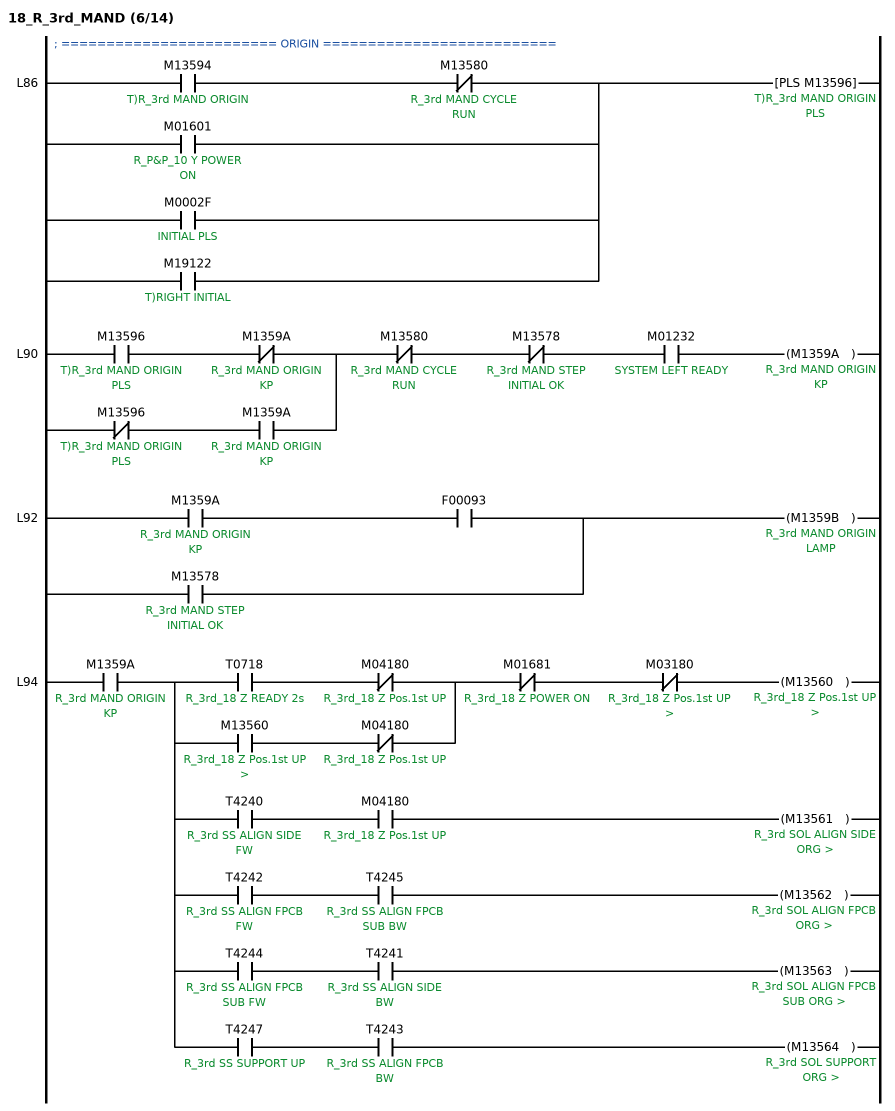
[picture p168: 18_R_3rd_MAND rungs L86-L94]
// ======================== ORIGIN ==========================
; L86
LOAD      M13594	// T)R_3rd MAND ORIGIN
AND NOT   M13580	// R_3rd MAND CYCLE RUN
OR        M01601	// R_P&P_10 Y POWER ON
OR        M0002F	// INITIAL PLS
OR        M19122	// T)RIGHT INITIAL
OUTP      M13596	// T)R_3rd MAND ORIGIN PLS
; L90
LOAD      M13596	// T)R_3rd MAND ORIGIN PLS
AND NOT   M1359A	// R_3rd MAND ORIGIN KP
LOAD NOT  M13596	// T)R_3rd MAND ORIGIN PLS
AND       M1359A	// R_3rd MAND ORIGIN KP
OR LOAD
AND NOT   M13580	// R_3rd MAND CYCLE RUN
AND NOT   M13578	// R_3rd MAND STEP INITIAL OK
AND       M01232	// SYSTEM LEFT READY
OUT       M1359A	// R_3rd MAND ORIGIN KP
; L92
LOAD      M1359A	// R_3rd MAND ORIGIN KP
AND       F00093
OR        M13578	// R_3rd MAND STEP INITIAL OK
OUT       M1359B	// R_3rd MAND ORIGIN LAMP
; L94
LOAD      M1359A	// R_3rd MAND ORIGIN KP
MPUSH
LOAD      T0718	// R_3rd_18 Z READY 2s
AND NOT   M04180	// R_3rd_18 Z Pos.1st UP
LOAD      M13560	// R_3rd_18 Z Pos.1st UP >
AND NOT   M04180	// R_3rd_18 Z Pos.1st UP
OR LOAD
AND LOAD
AND NOT   M01681	// R_3rd_18 Z POWER ON
AND NOT   M03180	// R_3rd_18 Z Pos.1st UP >
OUT       M13560	// R_3rd_18 Z Pos.1st UP >
MLOAD
AND       T4240	// R_3rd SS ALIGN SIDE FW
AND       M04180	// R_3rd_18 Z Pos.1st UP
OUT       M13561	// R_3rd SOL ALIGN SIDE ORG >
MLOAD
AND       T4242	// R_3rd SS ALIGN FPCB FW
AND       T4245	// R_3rd SS ALIGN FPCB SUB BW
OUT       M13562	// R_3rd SOL ALIGN FPCB ORG >
MLOAD
AND       T4244	// R_3rd SS ALIGN FPCB SUB FW
AND       T4241	// R_3rd SS ALIGN SIDE BW
OUT       M13563	// R_3rd SOL ALIGN FPCB SUB ORG >
MPOP
AND       T4247	// R_3rd SS SUPPORT UP
AND       T4243	// R_3rd SS ALIGN FPCB BW
OUT       M13564	// R_3rd SOL SUPPORT ORG >

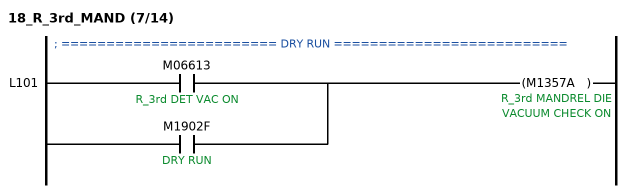
// ======================== DRY RUN ==========================
; L101
LOAD      M06613	// R_3rd DET VAC ON
OR        M1902F	// DRY RUN
OUT       M1357A	// R_3rd MANDREL DIE VACUUM CHECK ON

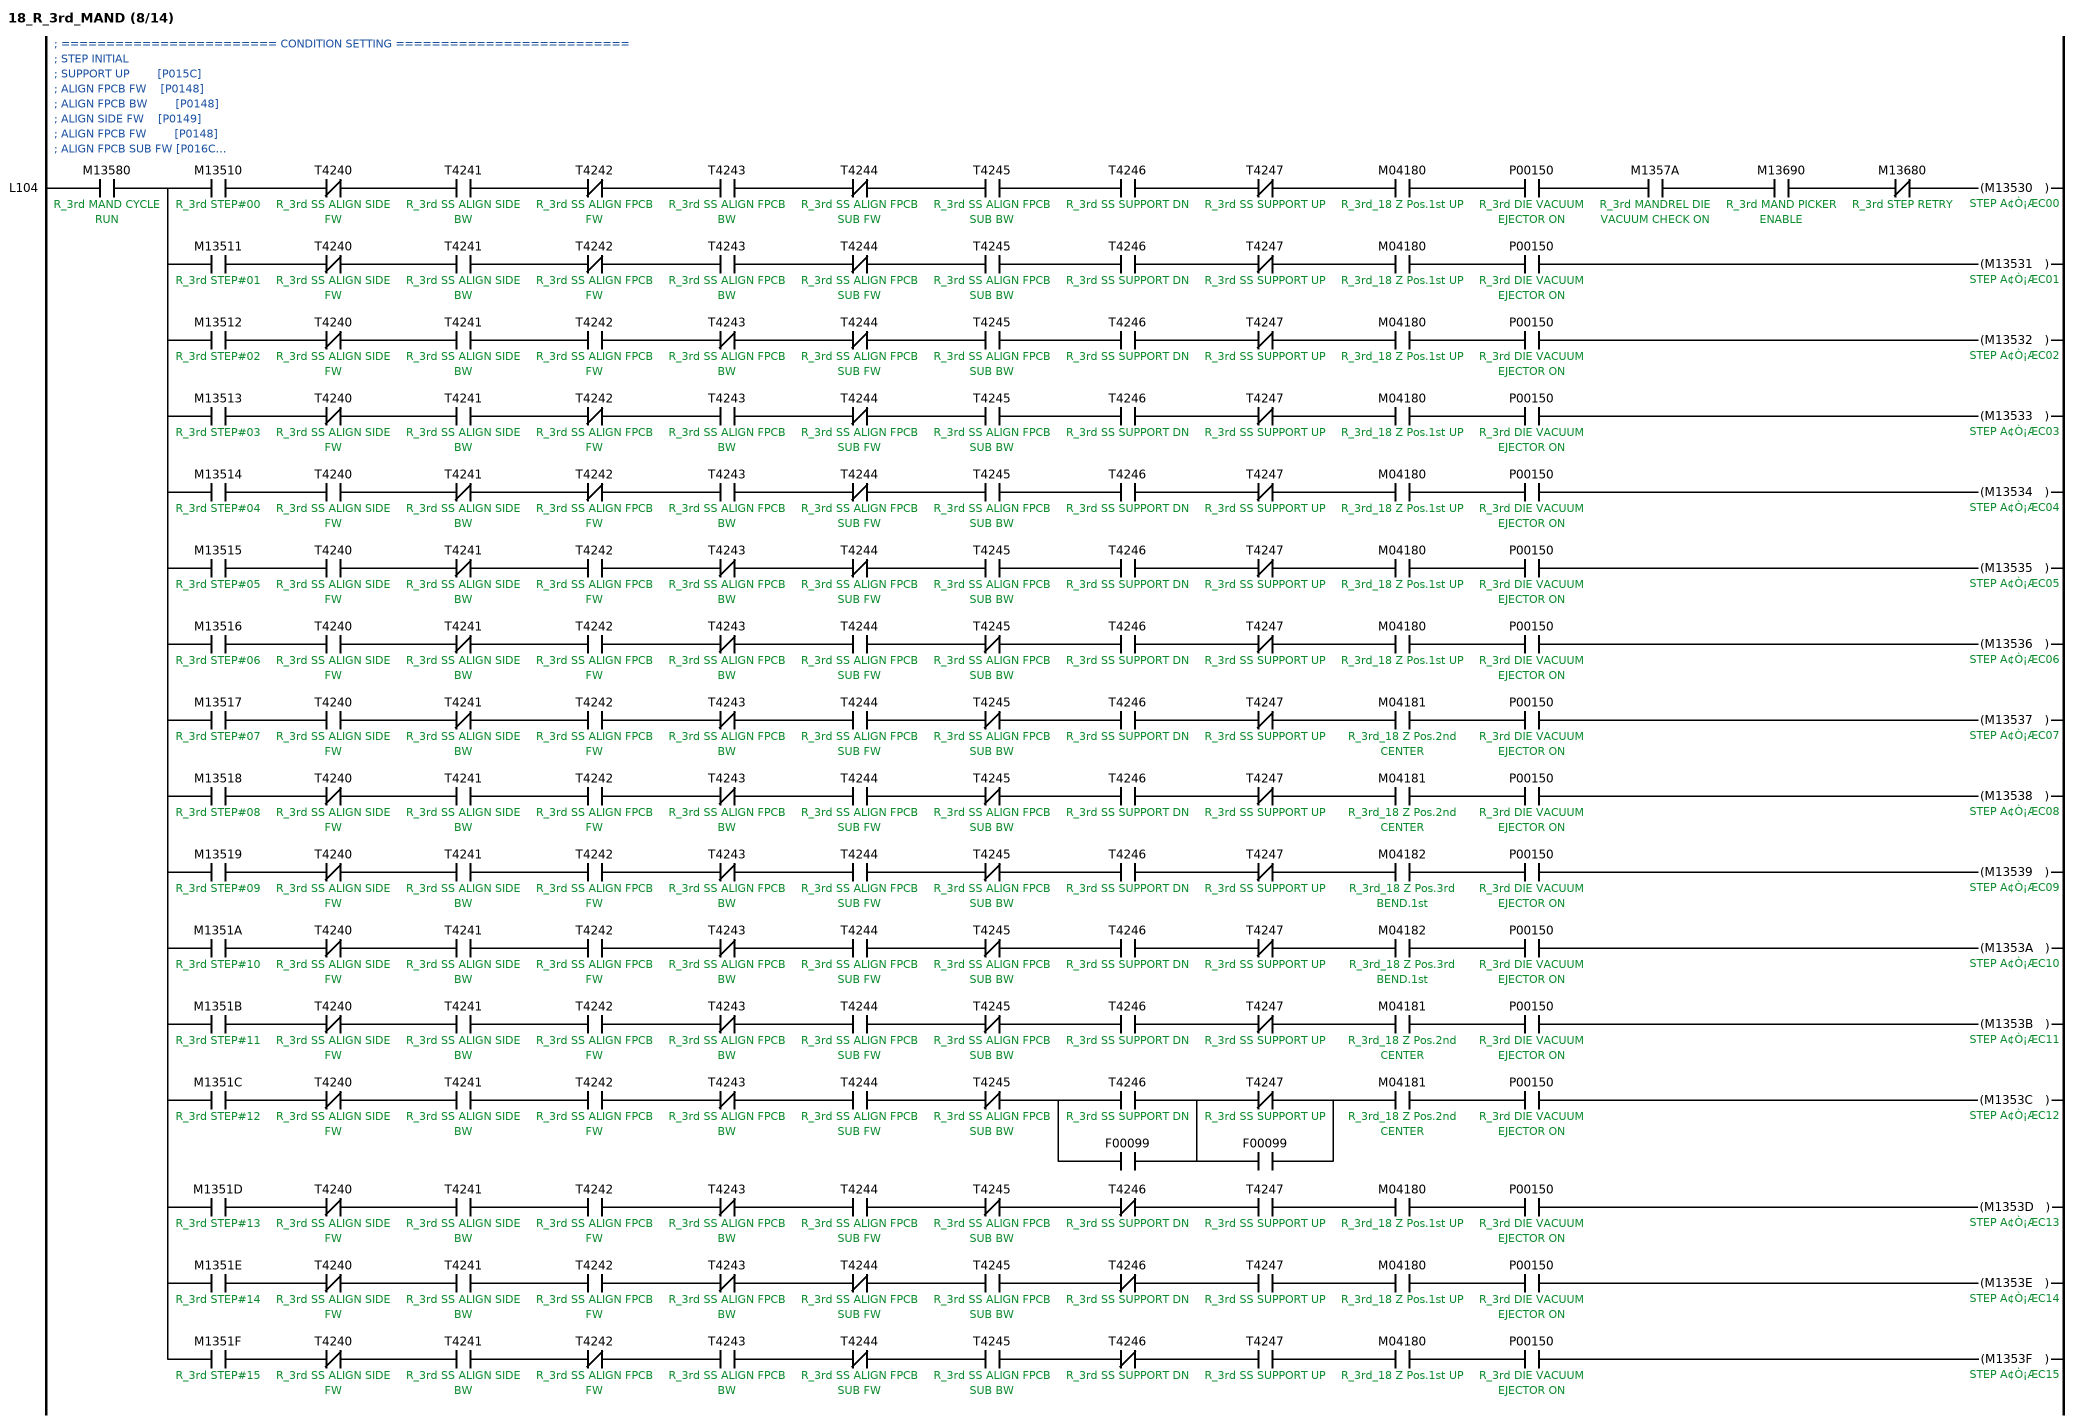
// ======================== CONDITION SETTING ==========================
; L104
LOAD      M13580	// R_3rd MAND CYCLE RUN
MPUSH
AND       M13510	// R_3rd STEP#00
AND NOT   T4240	// R_3rd SS ALIGN SIDE FW
AND       T4241	// R_3rd SS ALIGN SIDE BW
AND NOT   T4242	// R_3rd SS ALIGN FPCB FW
AND       T4243	// R_3rd SS ALIGN FPCB BW
AND NOT   T4244	// R_3rd SS ALIGN FPCB SUB FW
AND       T4245	// R_3rd SS ALIGN FPCB SUB BW
AND       T4246	// R_3rd SS SUPPORT DN
AND NOT   T4247	// R_3rd SS SUPPORT UP
AND       M04180	// R_3rd_18 Z Pos.1st UP
AND       P00150	// R_3rd DIE VACUUM EJECTOR ON
AND       M1357A	// R_3rd MANDREL DIE VACUUM CHECK ON
AND       M13690	// R_3rd MAND PICKER ENABLE
AND NOT   M13680	// R_3rd STEP RETRY
OUT       M13530	// STEP A¢Ò¡ÆC00
MLOAD
AND       M13511	// R_3rd STEP#01
AND NOT   T4240	// R_3rd SS ALIGN SIDE FW
AND       T4241	// R_3rd SS ALIGN SIDE BW
AND NOT   T4242	// R_3rd SS ALIGN FPCB FW
AND       T4243	// R_3rd SS ALIGN FPCB BW
AND NOT   T4244	// R_3rd SS ALIGN FPCB SUB FW
AND       T4245	// R_3rd SS ALIGN FPCB SUB BW
AND       T4246	// R_3rd SS SUPPORT DN
AND NOT   T4247	// R_3rd SS SUPPORT UP
AND       M04180	// R_3rd_18 Z Pos.1st UP
AND       P00150	// R_3rd DIE VACUUM EJECTOR ON
OUT       M13531	// STEP A¢Ò¡ÆC01
MLOAD
AND       M13512	// R_3rd STEP#02
AND NOT   T4240	// R_3rd SS ALIGN SIDE FW
AND       T4241	// R_3rd SS ALIGN SIDE BW
AND       T4242	// R_3rd SS ALIGN FPCB FW
AND NOT   T4243	// R_3rd SS ALIGN FPCB BW
AND NOT   T4244	// R_3rd SS ALIGN FPCB SUB FW
AND       T4245	// R_3rd SS ALIGN FPCB SUB BW
AND       T4246	// R_3rd SS SUPPORT DN
AND NOT   T4247	// R_3rd SS SUPPORT UP
AND       M04180	// R_3rd_18 Z Pos.1st UP
AND       P00150	// R_3rd DIE VACUUM EJECTOR ON
OUT       M13532	// STEP A¢Ò¡ÆC02
MLOAD
AND       M13513	// R_3rd STEP#03
AND NOT   T4240	// R_3rd SS ALIGN SIDE FW
AND       T4241	// R_3rd SS ALIGN SIDE BW
AND NOT   T4242	// R_3rd SS ALIGN FPCB FW
AND       T4243	// R_3rd SS ALIGN FPCB BW
AND NOT   T4244	// R_3rd SS ALIGN FPCB SUB FW
AND       T4245	// R_3rd SS ALIGN FPCB SUB BW
AND       T4246	// R_3rd SS SUPPORT DN
AND NOT   T4247	// R_3rd SS SUPPORT UP
AND       M04180	// R_3rd_18 Z Pos.1st UP
AND       P00150	// R_3rd DIE VACUUM EJECTOR ON
OUT       M13533	// STEP A¢Ò¡ÆC03
MLOAD
AND       M13514	// R_3rd STEP#04
AND       T4240	// R_3rd SS ALIGN SIDE FW
AND NOT   T4241	// R_3rd SS ALIGN SIDE BW
AND NOT   T4242	// R_3rd SS ALIGN FPCB FW
AND       T4243	// R_3rd SS ALIGN FPCB BW
AND NOT   T4244	// R_3rd SS ALIGN FPCB SUB FW
AND       T4245	// R_3rd SS ALIGN FPCB SUB BW
AND       T4246	// R_3rd SS SUPPORT DN
AND NOT   T4247	// R_3rd SS SUPPORT UP
AND       M04180	// R_3rd_18 Z Pos.1st UP
AND       P00150	// R_3rd DIE VACUUM EJECTOR ON
OUT       M13534	// STEP A¢Ò¡ÆC04
MLOAD
AND       M13515	// R_3rd STEP#05
AND       T4240	// R_3rd SS ALIGN SIDE FW
AND NOT   T4241	// R_3rd SS ALIGN SIDE BW
AND       T4242	// R_3rd SS ALIGN FPCB FW
AND NOT   T4243	// R_3rd SS ALIGN FPCB BW
AND NOT   T4244	// R_3rd SS ALIGN FPCB SUB FW
AND       T4245	// R_3rd SS ALIGN FPCB SUB BW
AND       T4246	// R_3rd SS SUPPORT DN
AND NOT   T4247	// R_3rd SS SUPPORT UP
AND       M04180	// R_3rd_18 Z Pos.1st UP
AND       P00150	// R_3rd DIE VACUUM EJECTOR ON
OUT       M13535	// STEP A¢Ò¡ÆC05
MLOAD
AND       M13516	// R_3rd STEP#06
AND       T4240	// R_3rd SS ALIGN SIDE FW
AND NOT   T4241	// R_3rd SS ALIGN SIDE BW
AND       T4242	// R_3rd SS ALIGN FPCB FW
AND NOT   T4243	// R_3rd SS ALIGN FPCB BW
AND       T4244	// R_3rd SS ALIGN FPCB SUB FW
AND NOT   T4245	// R_3rd SS ALIGN FPCB SUB BW
AND       T4246	// R_3rd SS SUPPORT DN
AND NOT   T4247	// R_3rd SS SUPPORT UP
AND       M04180	// R_3rd_18 Z Pos.1st UP
AND       P00150	// R_3rd DIE VACUUM EJECTOR ON
OUT       M13536	// STEP A¢Ò¡ÆC06
MLOAD
AND       M13517	// R_3rd STEP#07
AND       T4240	// R_3rd SS ALIGN SIDE FW
AND NOT   T4241	// R_3rd SS ALIGN SIDE BW
AND       T4242	// R_3rd SS ALIGN FPCB FW
AND NOT   T4243	// R_3rd SS ALIGN FPCB BW
AND       T4244	// R_3rd SS ALIGN FPCB SUB FW
AND NOT   T4245	// R_3rd SS ALIGN FPCB SUB BW
AND       T4246	// R_3rd SS SUPPORT DN
AND NOT   T4247	// R_3rd SS SUPPORT UP
AND       M04181	// R_3rd_18 Z Pos.2nd CENTER
AND       P00150	// R_3rd DIE VACUUM EJECTOR ON
OUT       M13537	// STEP A¢Ò¡ÆC07
MLOAD
AND       M13518	// R_3rd STEP#08
AND NOT   T4240	// R_3rd SS ALIGN SIDE FW
AND       T4241	// R_3rd SS ALIGN SIDE BW
AND       T4242	// R_3rd SS ALIGN FPCB FW
AND NOT   T4243	// R_3rd SS ALIGN FPCB BW
AND       T4244	// R_3rd SS ALIGN FPCB SUB FW
AND NOT   T4245	// R_3rd SS ALIGN FPCB SUB BW
AND       T4246	// R_3rd SS SUPPORT DN
AND NOT   T4247	// R_3rd SS SUPPORT UP
AND       M04181	// R_3rd_18 Z Pos.2nd CENTER
AND       P00150	// R_3rd DIE VACUUM EJECTOR ON
OUT       M13538	// STEP A¢Ò¡ÆC08
MLOAD
AND       M13519	// R_3rd STEP#09
AND NOT   T4240	// R_3rd SS ALIGN SIDE FW
AND       T4241	// R_3rd SS ALIGN SIDE BW
AND       T4242	// R_3rd SS ALIGN FPCB FW
AND NOT   T4243	// R_3rd SS ALIGN FPCB BW
AND       T4244	// R_3rd SS ALIGN FPCB SUB FW
AND NOT   T4245	// R_3rd SS ALIGN FPCB SUB BW
AND       T4246	// R_3rd SS SUPPORT DN
AND NOT   T4247	// R_3rd SS SUPPORT UP
AND       M04182	// R_3rd_18 Z Pos.3rd BEND.1st
AND       P00150	// R_3rd DIE VACUUM EJECTOR ON
OUT       M13539	// STEP A¢Ò¡ÆC09
MLOAD
AND       M1351A	// R_3rd STEP#10
AND NOT   T4240	// R_3rd SS ALIGN SIDE FW
AND       T4241	// R_3rd SS ALIGN SIDE BW
AND       T4242	// R_3rd SS ALIGN FPCB FW
AND NOT   T4243	// R_3rd SS ALIGN FPCB BW
AND       T4244	// R_3rd SS ALIGN FPCB SUB FW
AND NOT   T4245	// R_3rd SS ALIGN FPCB SUB BW
AND       T4246	// R_3rd SS SUPPORT DN
AND NOT   T4247	// R_3rd SS SUPPORT UP
AND       M04182	// R_3rd_18 Z Pos.3rd BEND.1st
AND       P00150	// R_3rd DIE VACUUM EJECTOR ON
OUT       M1353A	// STEP A¢Ò¡ÆC10
MLOAD
AND       M1351B	// R_3rd STEP#11
AND NOT   T4240	// R_3rd SS ALIGN SIDE FW
AND       T4241	// R_3rd SS ALIGN SIDE BW
AND       T4242	// R_3rd SS ALIGN FPCB FW
AND NOT   T4243	// R_3rd SS ALIGN FPCB BW
AND       T4244	// R_3rd SS ALIGN FPCB SUB FW
AND NOT   T4245	// R_3rd SS ALIGN FPCB SUB BW
AND       T4246	// R_3rd SS SUPPORT DN
AND NOT   T4247	// R_3rd SS SUPPORT UP
AND       M04181	// R_3rd_18 Z Pos.2nd CENTER
AND       P00150	// R_3rd DIE VACUUM EJECTOR ON
OUT       M1353B	// STEP A¢Ò¡ÆC11
MLOAD
AND       M1351C	// R_3rd STEP#12
AND NOT   T4240	// R_3rd SS ALIGN SIDE FW
AND       T4241	// R_3rd SS ALIGN SIDE BW
AND       T4242	// R_3rd SS ALIGN FPCB FW
AND NOT   T4243	// R_3rd SS ALIGN FPCB BW
AND       T4244	// R_3rd SS ALIGN FPCB SUB FW
AND NOT   T4245	// R_3rd SS ALIGN FPCB SUB BW
LOAD      T4246	// R_3rd SS SUPPORT DN
OR        F00099
AND LOAD
LOAD NOT  T4247	// R_3rd SS SUPPORT UP
OR        F00099
AND LOAD
AND       M04181	// R_3rd_18 Z Pos.2nd CENTER
AND       P00150	// R_3rd DIE VACUUM EJECTOR ON
OUT       M1353C	// STEP A¢Ò¡ÆC12
MLOAD
AND       M1351D	// R_3rd STEP#13
AND NOT   T4240	// R_3rd SS ALIGN SIDE FW
AND       T4241	// R_3rd SS ALIGN SIDE BW
AND       T4242	// R_3rd SS ALIGN FPCB FW
AND NOT   T4243	// R_3rd SS ALIGN FPCB BW
AND       T4244	// R_3rd SS ALIGN FPCB SUB FW
AND NOT   T4245	// R_3rd SS ALIGN FPCB SUB BW
AND NOT   T4246	// R_3rd SS SUPPORT DN
AND       T4247	// R_3rd SS SUPPORT UP
AND       M04180	// R_3rd_18 Z Pos.1st UP
AND       P00150	// R_3rd DIE VACUUM EJECTOR ON
OUT       M1353D	// STEP A¢Ò¡ÆC13
MLOAD
AND       M1351E	// R_3rd STEP#14
AND NOT   T4240	// R_3rd SS ALIGN SIDE FW
AND       T4241	// R_3rd SS ALIGN SIDE BW
AND       T4242	// R_3rd SS ALIGN FPCB FW
AND NOT   T4243	// R_3rd SS ALIGN FPCB BW
AND NOT   T4244	// R_3rd SS ALIGN FPCB SUB FW
AND       T4245	// R_3rd SS ALIGN FPCB SUB BW
AND NOT   T4246	// R_3rd SS SUPPORT DN
AND       T4247	// R_3rd SS SUPPORT UP
AND       M04180	// R_3rd_18 Z Pos.1st UP
AND       P00150	// R_3rd DIE VACUUM EJECTOR ON
OUT       M1353E	// STEP A¢Ò¡ÆC14
MPOP
AND       M1351F	// R_3rd STEP#15
AND NOT   T4240	// R_3rd SS ALIGN SIDE FW
AND       T4241	// R_3rd SS ALIGN SIDE BW
AND NOT   T4242	// R_3rd SS ALIGN FPCB FW
AND       T4243	// R_3rd SS ALIGN FPCB BW
AND NOT   T4244	// R_3rd SS ALIGN FPCB SUB FW
AND       T4245	// R_3rd SS ALIGN FPCB SUB BW
AND NOT   T4246	// R_3rd SS SUPPORT DN
AND       T4247	// R_3rd SS SUPPORT UP
AND       M04180	// R_3rd_18 Z Pos.1st UP
AND       P00150	// R_3rd DIE VACUUM EJECTOR ON
OUT       M1353F	// STEP A¢Ò¡ÆC15
// output comment: STEP INITIAL
// output comment: SUPPORT UP        [P015C]
// output comment: ALIGN FPCB FW    [P0148]
// output comment: ALIGN FPCB BW        [P0148]
// output comment: ALIGN SIDE FW    [P0149]
// output comment: ALIGN FPCB FW        [P0148]
// output comment: ALIGN FPCB SUB FW [P016C]
// output comment: R_3rd_18 Z Pos.2nd CENTER >
// output comment: ALIGN SIDE BW      [P0149]
// output comment: R_3rd_18 Z Pos.3rd BEND.1st >
// output comment: SUPPORT DN      [P015C]
// output comment: R_3rd_18 Z Pos.2nd CENTER >
// output comment: R_3rd_18 Z Pos.1st      UP >
// output comment: ALIGN FPCB SUB BW [P012D]
// output comment: ALIGN FPCB BW    [P0148]

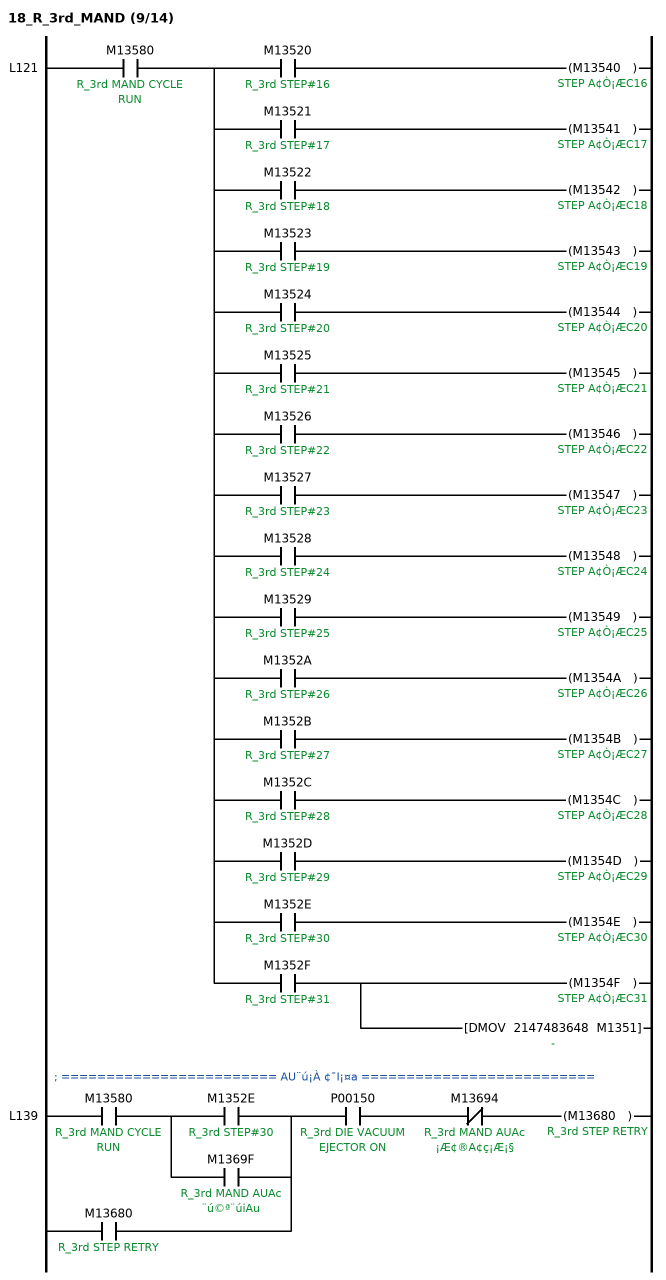
; L121
LOAD      M13580	// R_3rd MAND CYCLE RUN
MPUSH
AND       M13520	// R_3rd STEP#16
OUT       M13540	// STEP A¢Ò¡ÆC16
MLOAD
AND       M13521	// R_3rd STEP#17
OUT       M13541	// STEP A¢Ò¡ÆC17
MLOAD
AND       M13522	// R_3rd STEP#18
OUT       M13542	// STEP A¢Ò¡ÆC18
MLOAD
AND       M13523	// R_3rd STEP#19
OUT       M13543	// STEP A¢Ò¡ÆC19
MLOAD
AND       M13524	// R_3rd STEP#20
OUT       M13544	// STEP A¢Ò¡ÆC20
MLOAD
AND       M13525	// R_3rd STEP#21
OUT       M13545	// STEP A¢Ò¡ÆC21
MLOAD
AND       M13526	// R_3rd STEP#22
OUT       M13546	// STEP A¢Ò¡ÆC22
MLOAD
AND       M13527	// R_3rd STEP#23
OUT       M13547	// STEP A¢Ò¡ÆC23
MLOAD
AND       M13528	// R_3rd STEP#24
OUT       M13548	// STEP A¢Ò¡ÆC24
MLOAD
AND       M13529	// R_3rd STEP#25
OUT       M13549	// STEP A¢Ò¡ÆC25
MLOAD
AND       M1352A	// R_3rd STEP#26
OUT       M1354A	// STEP A¢Ò¡ÆC26
MLOAD
AND       M1352B	// R_3rd STEP#27
OUT       M1354B	// STEP A¢Ò¡ÆC27
MLOAD
AND       M1352C	// R_3rd STEP#28
OUT       M1354C	// STEP A¢Ò¡ÆC28
MLOAD
AND       M1352D	// R_3rd STEP#29
OUT       M1354D	// STEP A¢Ò¡ÆC29
MLOAD
AND       M1352E	// R_3rd STEP#30
OUT       M1354E	// STEP A¢Ò¡ÆC30
MPOP
AND       M1352F	// R_3rd STEP#31
OUT       M1354F	// STEP A¢Ò¡ÆC31
DMOV      2147483648 M1351	// -
// ======================== AU¨ú¡À ¢¯I¡¤a ==========================
; L139
LOAD      M13580	// R_3rd MAND CYCLE RUN
LOAD      M1352E	// R_3rd STEP#30
OR        M1369F	// R_3rd MAND AUAc ¨ú©ª¨úiAu
AND LOAD
OR        M13680	// R_3rd STEP RETRY
AND       P00150	// R_3rd DIE VACUUM EJECTOR ON
AND NOT   M13694	// R_3rd MAND AUAc ¡Æ¢®A¢ç¡Æ¡§
OUT       M13680	// R_3rd STEP RETRY

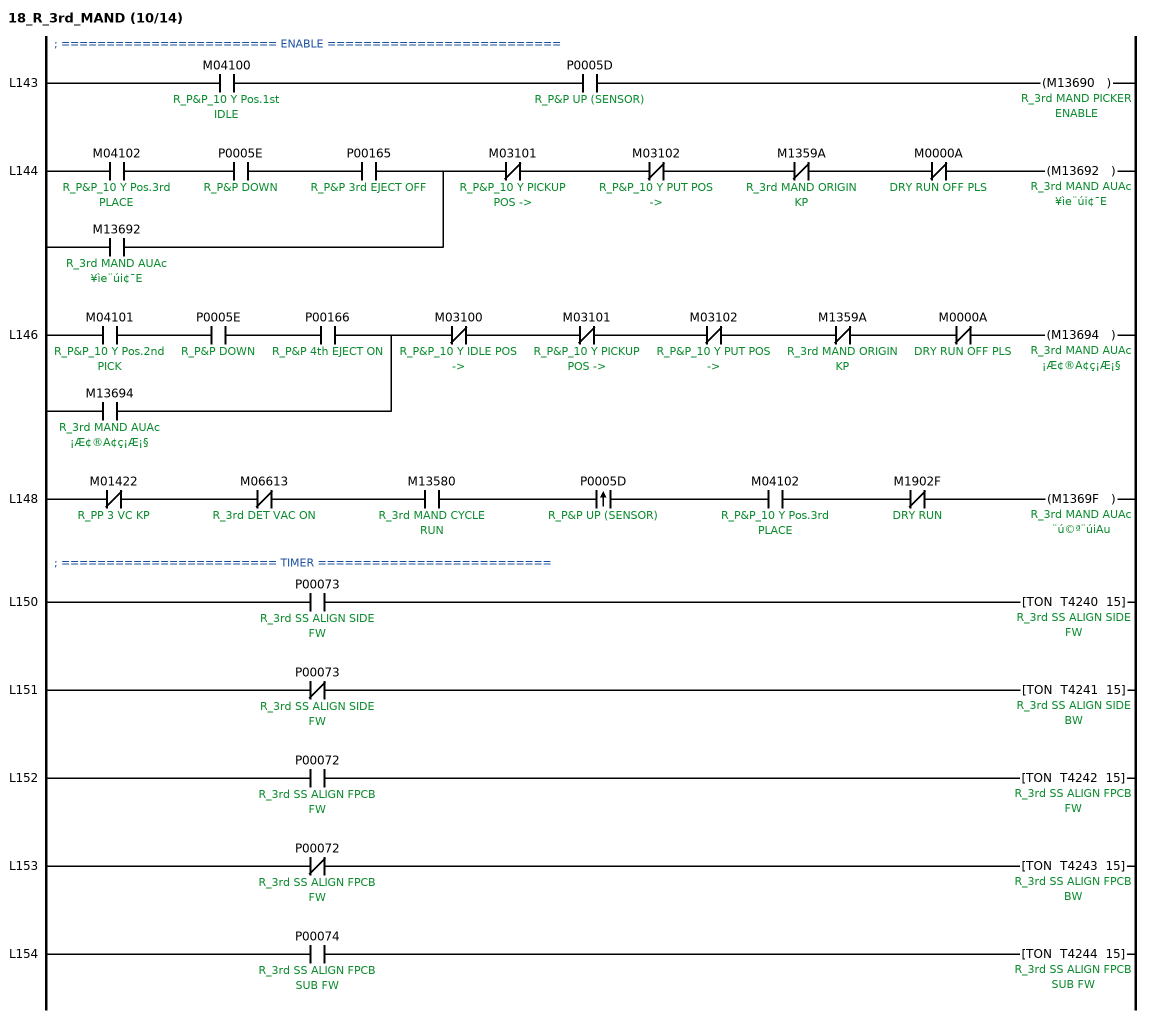
// ======================== ENABLE ==========================
; L143
LOAD      M04100	// R_P&P_10 Y Pos.1st IDLE
AND       P0005D	// R_P&P UP (SENSOR)
OUT       M13690	// R_3rd MAND PICKER ENABLE
; L144
LOAD      M04102	// R_P&P_10 Y Pos.3rd PLACE
AND       P0005E	// R_P&P DOWN
AND       P00165	// R_P&P 3rd EJECT OFF
OR        M13692	// R_3rd MAND AUAc ¥ìe¨úi¢¯E
AND NOT   M03101	// R_P&P_10 Y PICKUP POS ->
AND NOT   M03102	// R_P&P_10 Y PUT POS ->
AND NOT   M1359A	// R_3rd MAND ORIGIN KP
AND NOT   M0000A	// DRY RUN OFF PLS
OUT       M13692	// R_3rd MAND AUAc ¥ìe¨úi¢¯E
; L146
LOAD      M04101	// R_P&P_10 Y Pos.2nd PICK
AND       P0005E	// R_P&P DOWN
AND       P00166	// R_P&P 4th EJECT ON
OR        M13694	// R_3rd MAND AUAc ¡Æ¢®A¢ç¡Æ¡§
AND NOT   M03100	// R_P&P_10 Y IDLE POS ->
AND NOT   M03101	// R_P&P_10 Y PICKUP POS ->
AND NOT   M03102	// R_P&P_10 Y PUT POS ->
AND NOT   M1359A	// R_3rd MAND ORIGIN KP
AND NOT   M0000A	// DRY RUN OFF PLS
OUT       M13694	// R_3rd MAND AUAc ¡Æ¢®A¢ç¡Æ¡§
; L148
LOAD NOT  M01422	// R_PP 3 VC KP
AND NOT   M06613	// R_3rd DET VAC ON
AND       M13580	// R_3rd MAND CYCLE RUN
ANDP      P0005D	// R_P&P UP (SENSOR)
AND       M04102	// R_P&P_10 Y Pos.3rd PLACE
AND NOT   M1902F	// DRY RUN
OUT       M1369F	// R_3rd MAND AUAc ¨ú©ª¨úiAu
// ======================== TIMER ==========================
; L150
LOAD      P00073	// R_3rd SS ALIGN SIDE FW
TON       T4240 15	// R_3rd SS ALIGN SIDE FW
; L151
LOAD NOT  P00073	// R_3rd SS ALIGN SIDE FW
TON       T4241 15	// R_3rd SS ALIGN SIDE BW
; L152
LOAD      P00072	// R_3rd SS ALIGN FPCB FW
TON       T4242 15	// R_3rd SS ALIGN FPCB FW
; L153
LOAD NOT  P00072	// R_3rd SS ALIGN FPCB FW
TON       T4243 15	// R_3rd SS ALIGN FPCB BW
; L154
LOAD      P00074	// R_3rd SS ALIGN FPCB SUB FW
TON       T4244 15	// R_3rd SS ALIGN FPCB SUB FW

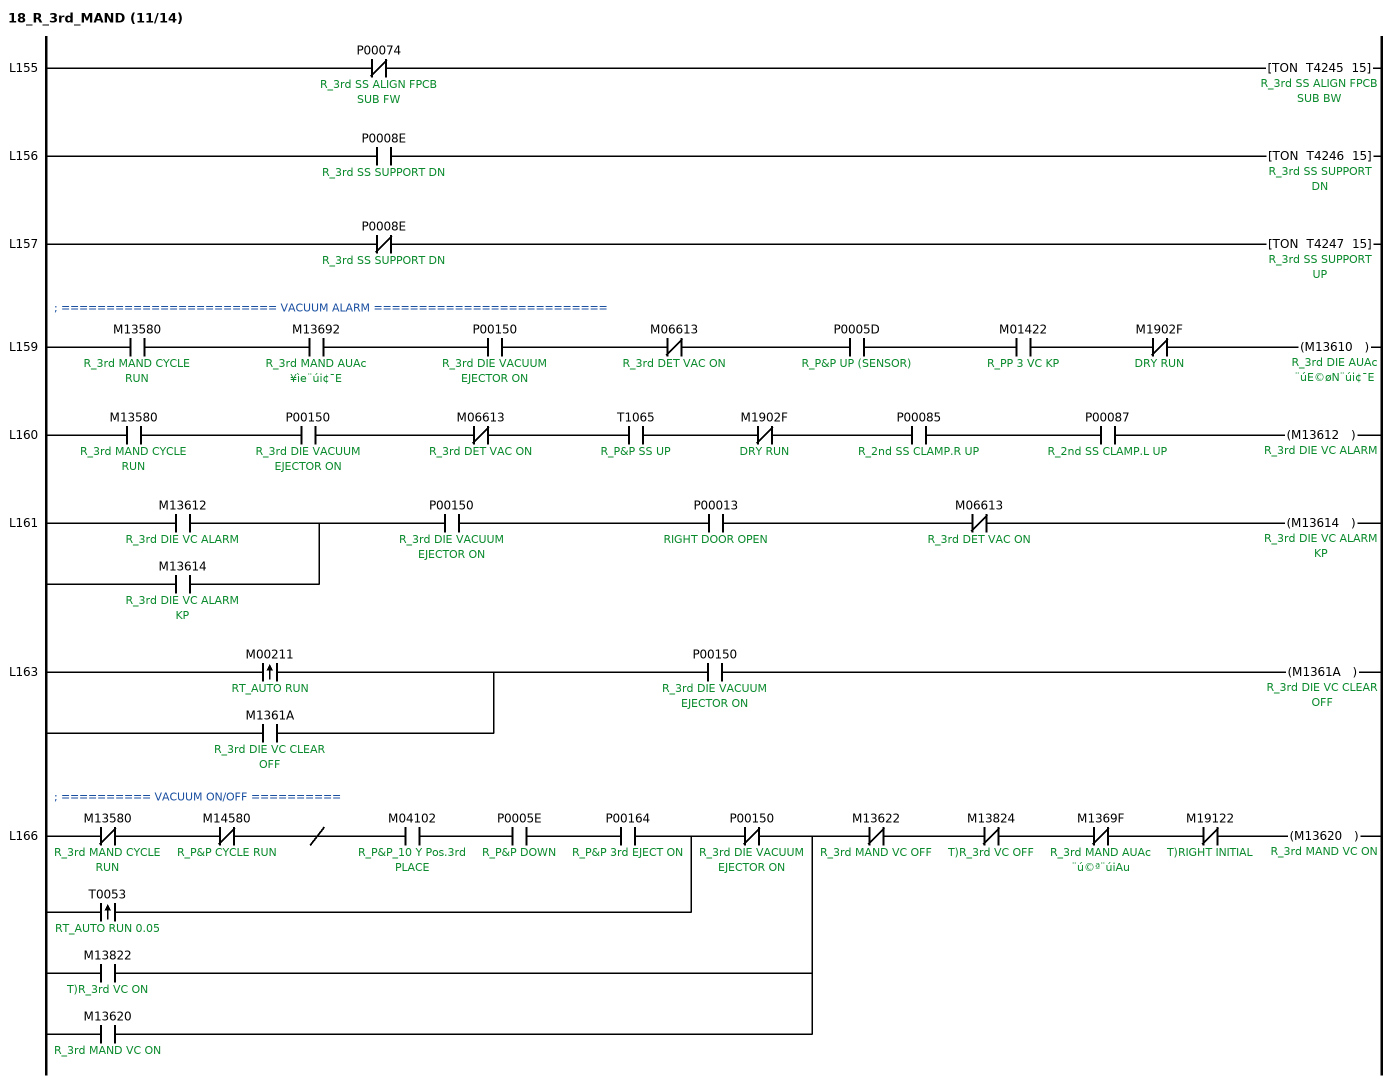
; L155
LOAD NOT  P00074	// R_3rd SS ALIGN FPCB SUB FW
TON       T4245 15	// R_3rd SS ALIGN FPCB SUB BW
; L156
LOAD      P0008E	// R_3rd SS SUPPORT DN
TON       T4246 15	// R_3rd SS SUPPORT DN
; L157
LOAD NOT  P0008E	// R_3rd SS SUPPORT DN
TON       T4247 15	// R_3rd SS SUPPORT UP
// ======================== VACUUM ALARM ==========================
; L159
LOAD      M13580	// R_3rd MAND CYCLE RUN
AND       M13692	// R_3rd MAND AUAc ¥ìe¨úi¢¯E
AND       P00150	// R_3rd DIE VACUUM EJECTOR ON
AND NOT   M06613	// R_3rd DET VAC ON
AND       P0005D	// R_P&P UP (SENSOR)
AND       M01422	// R_PP 3 VC KP
AND NOT   M1902F	// DRY RUN
OUT       M13610	// R_3rd DIE AUAc ¨úE©øN¨úi¢¯E
; L160
LOAD      M13580	// R_3rd MAND CYCLE RUN
AND       P00150	// R_3rd DIE VACUUM EJECTOR ON
AND NOT   M06613	// R_3rd DET VAC ON
AND       T1065	// R_P&P SS UP
AND NOT   M1902F	// DRY RUN
AND       P00085	// R_2nd SS CLAMP.R UP
AND       P00087	// R_2nd SS CLAMP.L UP
OUT       M13612	// R_3rd DIE VC ALARM
; L161
LOAD      M13612	// R_3rd DIE VC ALARM
OR        M13614	// R_3rd DIE VC ALARM KP
AND       P00150	// R_3rd DIE VACUUM EJECTOR ON
AND       P00013	// RIGHT DOOR OPEN
AND NOT   M06613	// R_3rd DET VAC ON
OUT       M13614	// R_3rd DIE VC ALARM KP
; L163
LOADP     M00211	// RT_AUTO RUN
OR        M1361A	// R_3rd DIE VC CLEAR OFF
AND       P00150	// R_3rd DIE VACUUM EJECTOR ON
OUT       M1361A	// R_3rd DIE VC CLEAR OFF
// ========== VACUUM ON/OFF ==========
; L166
LOAD NOT  M13580	// R_3rd MAND CYCLE RUN
AND NOT   M14580	// R_P&P CYCLE RUN
NOT
AND       M04102	// R_P&P_10 Y Pos.3rd PLACE
AND       P0005E	// R_P&P DOWN
AND       P00164	// R_P&P 3rd EJECT ON
ORP       T0053	// RT_AUTO RUN 0.05
AND NOT   P00150	// R_3rd DIE VACUUM EJECTOR ON
OR        M13822	// T)R_3rd VC ON
OR        M13620	// R_3rd MAND VC ON
AND NOT   M13622	// R_3rd MAND VC OFF
AND NOT   M13824	// T)R_3rd VC OFF
AND NOT   M1369F	// R_3rd MAND AUAc ¨ú©ª¨úiAu
AND NOT   M19122	// T)RIGHT INITIAL
OUT       M13620	// R_3rd MAND VC ON

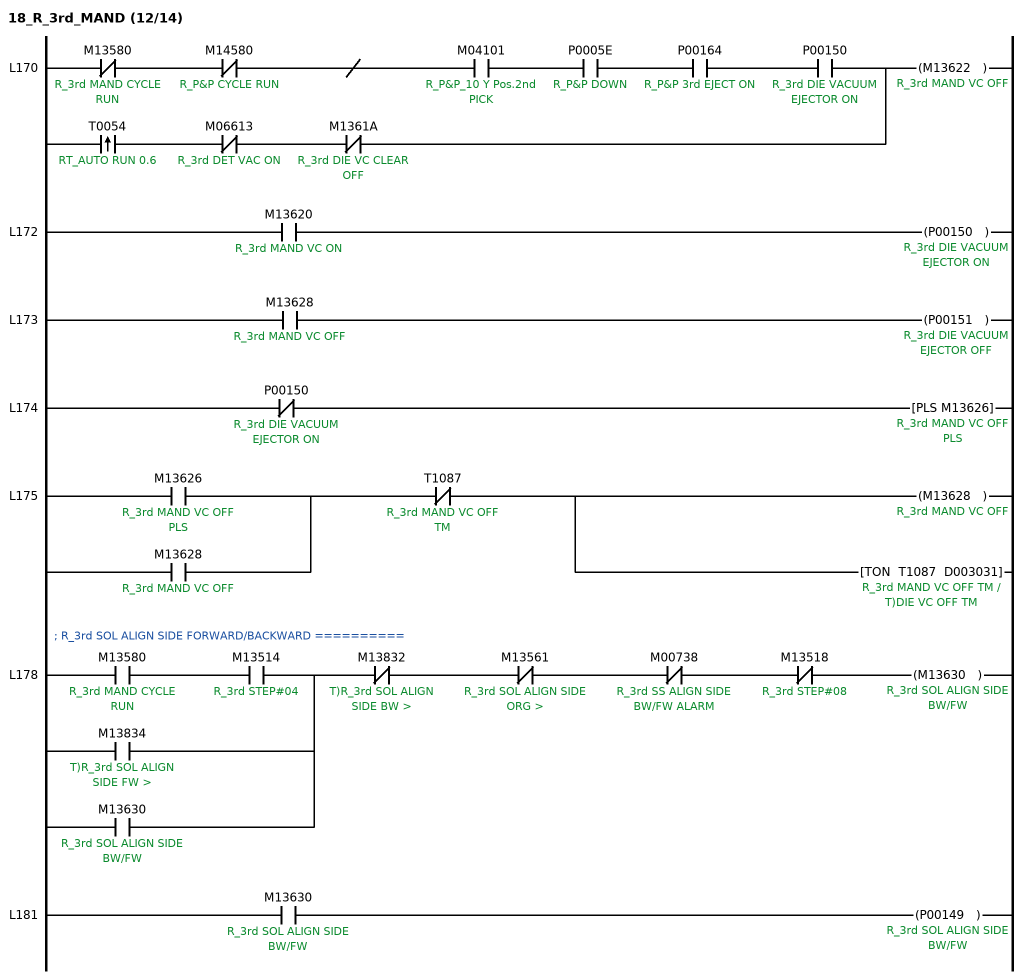
; L170
LOAD NOT  M13580	// R_3rd MAND CYCLE RUN
AND NOT   M14580	// R_P&P CYCLE RUN
NOT
AND       M04101	// R_P&P_10 Y Pos.2nd PICK
AND       P0005E	// R_P&P DOWN
AND       P00164	// R_P&P 3rd EJECT ON
AND       P00150	// R_3rd DIE VACUUM EJECTOR ON
LOADP     T0054	// RT_AUTO RUN 0.6
AND NOT   M06613	// R_3rd DET VAC ON
AND NOT   M1361A	// R_3rd DIE VC CLEAR OFF
OR LOAD
OUT       M13622	// R_3rd MAND VC OFF
; L172
LOAD      M13620	// R_3rd MAND VC ON
OUT       P00150	// R_3rd DIE VACUUM EJECTOR ON
; L173
LOAD      M13628	// R_3rd MAND VC OFF
OUT       P00151	// R_3rd DIE VACUUM EJECTOR OFF
; L174
LOAD NOT  P00150	// R_3rd DIE VACUUM EJECTOR ON
OUTP      M13626	// R_3rd MAND VC OFF PLS
; L175
LOAD      M13626	// R_3rd MAND VC OFF PLS
OR        M13628	// R_3rd MAND VC OFF
AND NOT   T1087	// R_3rd MAND VC OFF TM
OUT       M13628	// R_3rd MAND VC OFF
TON       T1087 D003031	// R_3rd MAND VC OFF TM / T)DIE VC OFF TM
// R_3rd SOL ALIGN SIDE FORWARD/BACKWARD ==========
; L178
LOAD      M13580	// R_3rd MAND CYCLE RUN
AND       M13514	// R_3rd STEP#04
OR        M13834	// T)R_3rd SOL ALIGN SIDE FW >
OR        M13630	// R_3rd SOL ALIGN SIDE BW/FW
AND NOT   M13832	// T)R_3rd SOL ALIGN SIDE BW >
AND NOT   M13561	// R_3rd SOL ALIGN SIDE ORG >
AND NOT   M00738	// R_3rd SS ALIGN SIDE BW/FW ALARM
AND NOT   M13518	// R_3rd STEP#08
OUT       M13630	// R_3rd SOL ALIGN SIDE BW/FW
; L181
LOAD      M13630	// R_3rd SOL ALIGN SIDE BW/FW
OUT       P00149	// R_3rd SOL ALIGN SIDE BW/FW

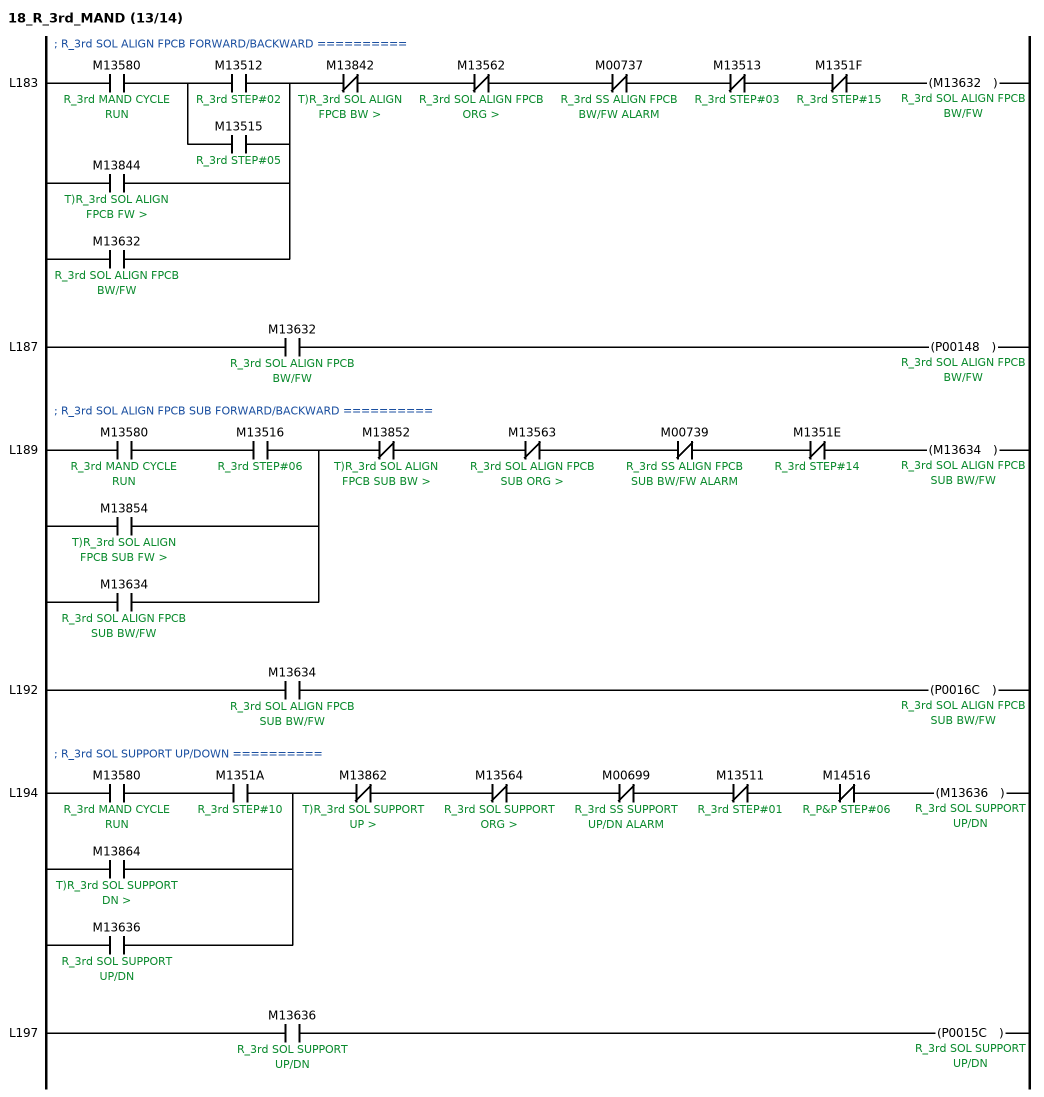
// R_3rd SOL ALIGN FPCB FORWARD/BACKWARD ==========
; L183
LOAD      M13580	// R_3rd MAND CYCLE RUN
LOAD      M13512	// R_3rd STEP#02
OR        M13515	// R_3rd STEP#05
AND LOAD
OR        M13844	// T)R_3rd SOL ALIGN FPCB FW >
OR        M13632	// R_3rd SOL ALIGN FPCB BW/FW
AND NOT   M13842	// T)R_3rd SOL ALIGN FPCB BW >
AND NOT   M13562	// R_3rd SOL ALIGN FPCB ORG >
AND NOT   M00737	// R_3rd SS ALIGN FPCB BW/FW ALARM
AND NOT   M13513	// R_3rd STEP#03
AND NOT   M1351F	// R_3rd STEP#15
OUT       M13632	// R_3rd SOL ALIGN FPCB BW/FW
; L187
LOAD      M13632	// R_3rd SOL ALIGN FPCB BW/FW
OUT       P00148	// R_3rd SOL ALIGN FPCB BW/FW
// R_3rd SOL ALIGN FPCB SUB FORWARD/BACKWARD ==========
; L189
LOAD      M13580	// R_3rd MAND CYCLE RUN
AND       M13516	// R_3rd STEP#06
OR        M13854	// T)R_3rd SOL ALIGN FPCB SUB FW >
OR        M13634	// R_3rd SOL ALIGN FPCB SUB BW/FW
AND NOT   M13852	// T)R_3rd SOL ALIGN FPCB SUB BW >
AND NOT   M13563	// R_3rd SOL ALIGN FPCB SUB ORG >
AND NOT   M00739	// R_3rd SS ALIGN FPCB SUB BW/FW ALARM
AND NOT   M1351E	// R_3rd STEP#14
OUT       M13634	// R_3rd SOL ALIGN FPCB SUB BW/FW
; L192
LOAD      M13634	// R_3rd SOL ALIGN FPCB SUB BW/FW
OUT       P0016C	// R_3rd SOL ALIGN FPCB SUB BW/FW
// R_3rd SOL SUPPORT UP/DOWN ==========
; L194
LOAD      M13580	// R_3rd MAND CYCLE RUN
AND       M1351A	// R_3rd STEP#10
OR        M13864	// T)R_3rd SOL SUPPORT DN >
OR        M13636	// R_3rd SOL SUPPORT UP/DN
AND NOT   M13862	// T)R_3rd SOL SUPPORT UP >
AND NOT   M13564	// R_3rd SOL SUPPORT ORG >
AND NOT   M00699	// R_3rd SS SUPPORT UP/DN ALARM
AND NOT   M13511	// R_3rd STEP#01
AND NOT   M14516	// R_P&P STEP#06
OUT       M13636	// R_3rd SOL SUPPORT UP/DN
; L197
LOAD      M13636	// R_3rd SOL SUPPORT UP/DN
OUT       P0015C	// R_3rd SOL SUPPORT UP/DN

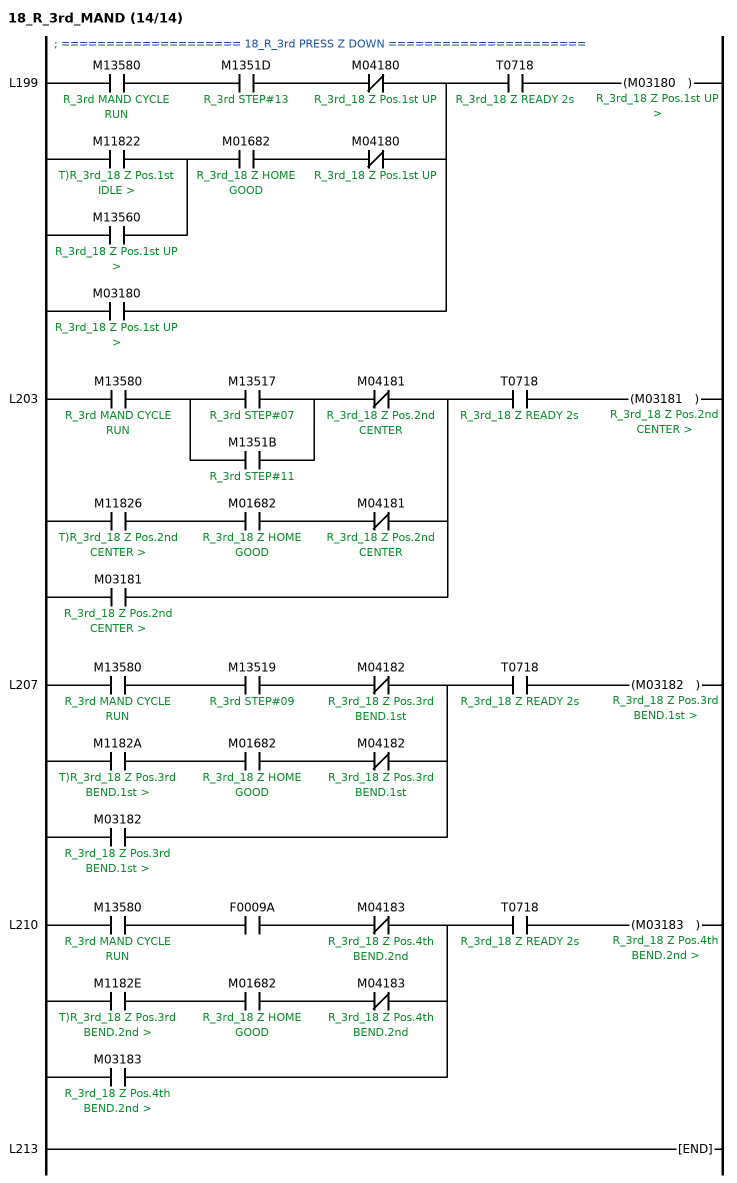
// ==================== 18_R_3rd PRESS Z DOWN ======================
; L199
LOAD      M13580	// R_3rd MAND CYCLE RUN
AND       M1351D	// R_3rd STEP#13
AND NOT   M04180	// R_3rd_18 Z Pos.1st UP
LOAD      M11822	// T)R_3rd_18 Z Pos.1st IDLE >
OR        M13560	// R_3rd_18 Z Pos.1st UP >
AND       M01682	// R_3rd_18 Z HOME GOOD
AND NOT   M04180	// R_3rd_18 Z Pos.1st UP
OR LOAD
OR        M03180	// R_3rd_18 Z Pos.1st UP >
AND       T0718	// R_3rd_18 Z READY 2s
OUT       M03180	// R_3rd_18 Z Pos.1st UP >
; L203
LOAD      M13580	// R_3rd MAND CYCLE RUN
LOAD      M13517	// R_3rd STEP#07
OR        M1351B	// R_3rd STEP#11
AND LOAD
AND NOT   M04181	// R_3rd_18 Z Pos.2nd CENTER
LOAD      M11826	// T)R_3rd_18 Z Pos.2nd CENTER >
AND       M01682	// R_3rd_18 Z HOME GOOD
AND NOT   M04181	// R_3rd_18 Z Pos.2nd CENTER
OR LOAD
OR        M03181	// R_3rd_18 Z Pos.2nd CENTER >
AND       T0718	// R_3rd_18 Z READY 2s
OUT       M03181	// R_3rd_18 Z Pos.2nd CENTER >
; L207
LOAD      M13580	// R_3rd MAND CYCLE RUN
AND       M13519	// R_3rd STEP#09
AND NOT   M04182	// R_3rd_18 Z Pos.3rd BEND.1st
LOAD      M1182A	// T)R_3rd_18 Z Pos.3rd BEND.1st >
AND       M01682	// R_3rd_18 Z HOME GOOD
AND NOT   M04182	// R_3rd_18 Z Pos.3rd BEND.1st
OR LOAD
OR        M03182	// R_3rd_18 Z Pos.3rd BEND.1st >
AND       T0718	// R_3rd_18 Z READY 2s
OUT       M03182	// R_3rd_18 Z Pos.3rd BEND.1st >
; L210
LOAD      M13580	// R_3rd MAND CYCLE RUN
AND       F0009A
AND NOT   M04183	// R_3rd_18 Z Pos.4th BEND.2nd
LOAD      M1182E	// T)R_3rd_18 Z Pos.3rd BEND.2nd >
AND       M01682	// R_3rd_18 Z HOME GOOD
AND NOT   M04183	// R_3rd_18 Z Pos.4th BEND.2nd
OR LOAD
OR        M03183	// R_3rd_18 Z Pos.4th BEND.2nd >
AND       T0718	// R_3rd_18 Z READY 2s
OUT       M03183	// R_3rd_18 Z Pos.4th BEND.2nd >
; L213
END

PROGRAM 19_R_TOOL (task: ¨ö¨¬A¥ì CA¡¤I¡¾¡¿¡¤¡Í)

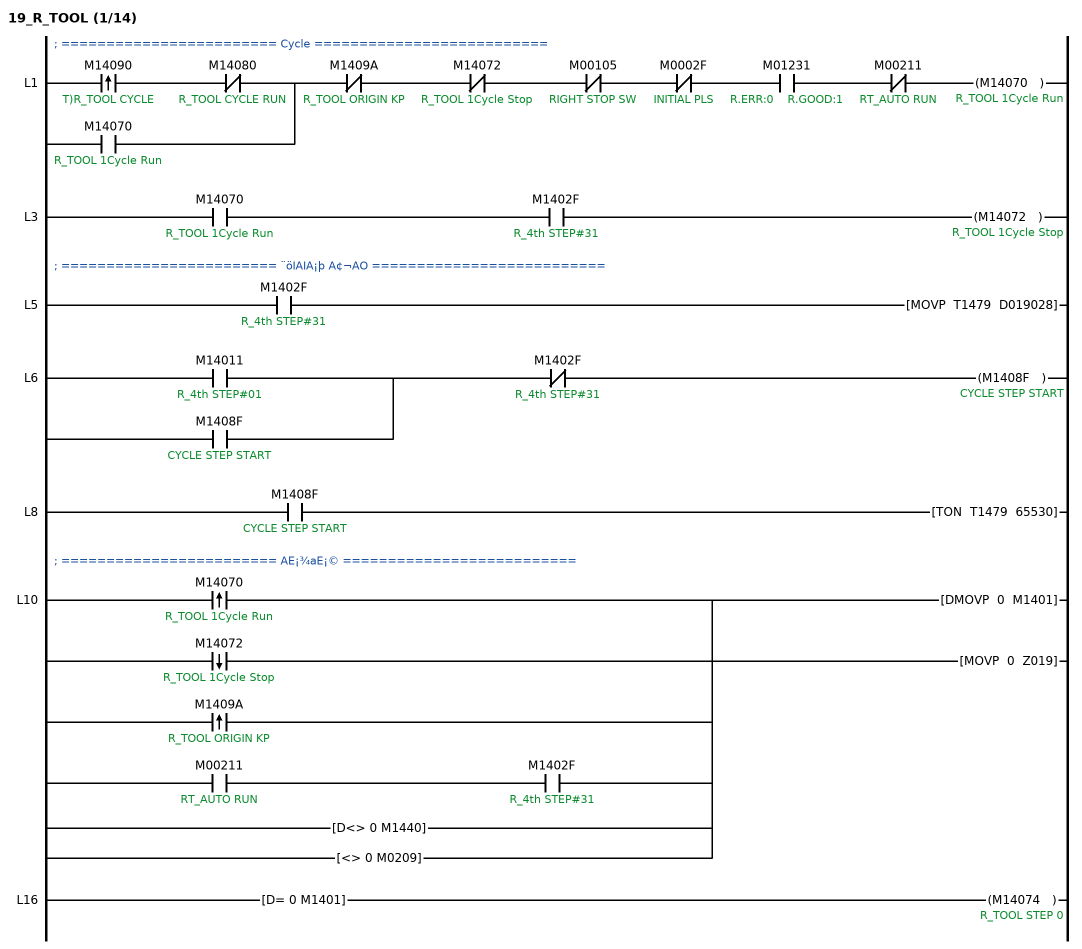
// ======================== Cycle ==========================
; L1
LOADP     M14090	// T)R_TOOL CYCLE
AND NOT   M14080	// R_TOOL CYCLE RUN
OR        M14070	// R_TOOL 1Cycle Run
AND NOT   M1409A	// R_TOOL ORIGIN KP
AND NOT   M14072	// R_TOOL 1Cycle Stop
AND NOT   M00105	// RIGHT STOP SW
AND NOT   M0002F	// INITIAL PLS
AND       M01231	// R.ERR:0    R.GOOD:1
AND NOT   M00211	// RT_AUTO RUN
OUT       M14070	// R_TOOL 1Cycle Run
; L3
LOAD      M14070	// R_TOOL 1Cycle Run
AND       M1402F	// R_4th STEP#31
OUT       M14072	// R_TOOL 1Cycle Stop
// ======================== ¨öIAIA¡þ A¢¬AO ==========================
; L5
LOAD      M1402F	// R_4th STEP#31
MOVP      T1479 D019028
; L6
LOAD      M14011	// R_4th STEP#01
OR        M1408F	// CYCLE STEP START
AND NOT   M1402F	// R_4th STEP#31
OUT       M1408F	// CYCLE STEP START
; L8
LOAD      M1408F	// CYCLE STEP START
TON       T1479 65530
// ======================== AE¡¾aE¡© ==========================
; L10
LOADP     M14070	// R_TOOL 1Cycle Run
ORN       M14072	// R_TOOL 1Cycle Stop
ORP       M1409A	// R_TOOL ORIGIN KP
LOAD      M00211	// RT_AUTO RUN
AND       M1402F	// R_4th STEP#31
OR LOAD
ORD<>     0 M1440
OR<>      0 M0209
DMOVP     0 M1401
MOVP      0 Z019
; L16
LOADD=    0 M1401
OUT       M14074	// R_TOOL STEP 0

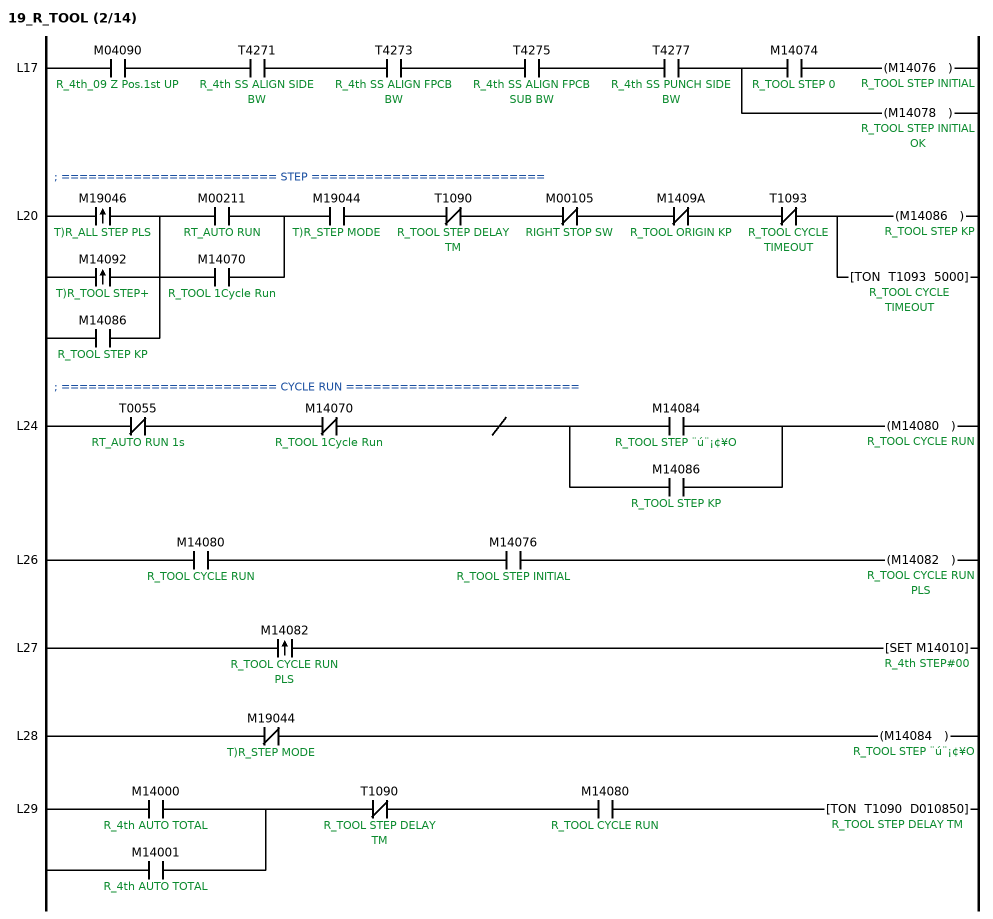
; L17
LOAD      M04090	// R_4th_09 Z Pos.1st UP
AND       T4271	// R_4th SS ALIGN SIDE BW
AND       T4273	// R_4th SS ALIGN FPCB BW
AND       T4275	// R_4th SS ALIGN FPCB SUB BW
AND       T4277	// R_4th SS PUNCH SIDE BW
MPUSH
AND       M14074	// R_TOOL STEP 0
OUT       M14076	// R_TOOL STEP INITIAL
MPOP
OUT       M14078	// R_TOOL STEP INITIAL OK
// ======================== STEP ==========================
; L20
LOADP     M19046	// T)R_ALL STEP PLS
ORP       M14092	// T)R_TOOL STEP+
OR        M14086	// R_TOOL STEP KP
LOAD      M00211	// RT_AUTO RUN
OR        M14070	// R_TOOL 1Cycle Run
AND LOAD
AND       M19044	// T)R_STEP MODE
AND NOT   T1090	// R_TOOL STEP DELAY TM
AND NOT   M00105	// RIGHT STOP SW
AND NOT   M1409A	// R_TOOL ORIGIN KP
AND NOT   T1093	// R_TOOL CYCLE TIMEOUT
OUT       M14086	// R_TOOL STEP KP
TON       T1093 5000	// R_TOOL CYCLE TIMEOUT
// ======================== CYCLE RUN ==========================
; L24
LOAD NOT  T0055	// RT_AUTO RUN 1s
AND NOT   M14070	// R_TOOL 1Cycle Run
NOT
LOAD      M14084	// R_TOOL STEP ¨ú¨¡¢¥O
OR        M14086	// R_TOOL STEP KP
AND LOAD
OUT       M14080	// R_TOOL CYCLE RUN
; L26
LOAD      M14080	// R_TOOL CYCLE RUN
AND       M14076	// R_TOOL STEP INITIAL
OUT       M14082	// R_TOOL CYCLE RUN PLS
; L27
LOADP     M14082	// R_TOOL CYCLE RUN PLS
SET       M14010	// R_4th STEP#00
; L28
LOAD NOT  M19044	// T)R_STEP MODE
OUT       M14084	// R_TOOL STEP ¨ú¨¡¢¥O
; L29
LOAD      M14000	// R_4th AUTO TOTAL
OR        M14001	// R_4th AUTO TOTAL
AND NOT   T1090	// R_TOOL STEP DELAY TM
AND       M14080	// R_TOOL CYCLE RUN
TON       T1090 D010850	// R_TOOL STEP DELAY TM

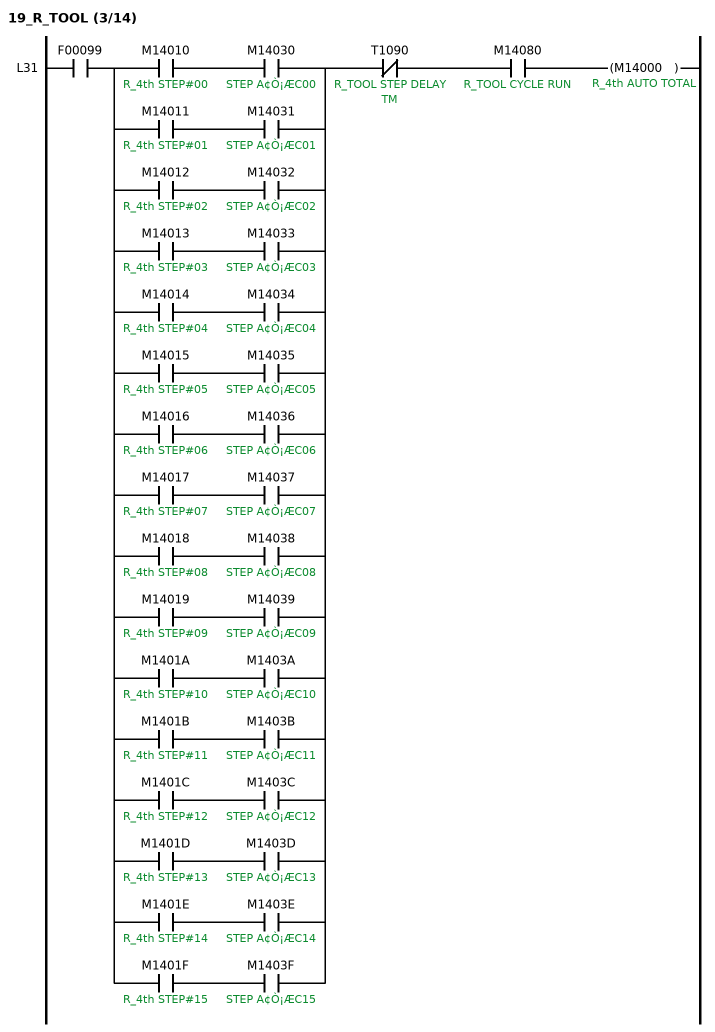
; L31
LOAD      F00099
LOAD      M14010	// R_4th STEP#00
AND       M14030	// STEP A¢Ò¡ÆC00
LOAD      M14011	// R_4th STEP#01
AND       M14031	// STEP A¢Ò¡ÆC01
OR LOAD
LOAD      M14012	// R_4th STEP#02
AND       M14032	// STEP A¢Ò¡ÆC02
OR LOAD
LOAD      M14013	// R_4th STEP#03
AND       M14033	// STEP A¢Ò¡ÆC03
OR LOAD
LOAD      M14014	// R_4th STEP#04
AND       M14034	// STEP A¢Ò¡ÆC04
OR LOAD
LOAD      M14015	// R_4th STEP#05
AND       M14035	// STEP A¢Ò¡ÆC05
OR LOAD
LOAD      M14016	// R_4th STEP#06
AND       M14036	// STEP A¢Ò¡ÆC06
OR LOAD
LOAD      M14017	// R_4th STEP#07
AND       M14037	// STEP A¢Ò¡ÆC07
OR LOAD
LOAD      M14018	// R_4th STEP#08
AND       M14038	// STEP A¢Ò¡ÆC08
OR LOAD
LOAD      M14019	// R_4th STEP#09
AND       M14039	// STEP A¢Ò¡ÆC09
OR LOAD
LOAD      M1401A	// R_4th STEP#10
AND       M1403A	// STEP A¢Ò¡ÆC10
OR LOAD
LOAD      M1401B	// R_4th STEP#11
AND       M1403B	// STEP A¢Ò¡ÆC11
OR LOAD
LOAD      M1401C	// R_4th STEP#12
AND       M1403C	// STEP A¢Ò¡ÆC12
OR LOAD
LOAD      M1401D	// R_4th STEP#13
AND       M1403D	// STEP A¢Ò¡ÆC13
OR LOAD
LOAD      M1401E	// R_4th STEP#14
AND       M1403E	// STEP A¢Ò¡ÆC14
OR LOAD
LOAD      M1401F	// R_4th STEP#15
AND       M1403F	// STEP A¢Ò¡ÆC15
OR LOAD
AND LOAD
AND NOT   T1090	// R_TOOL STEP DELAY TM
AND       M14080	// R_TOOL CYCLE RUN
OUT       M14000	// R_4th AUTO TOTAL

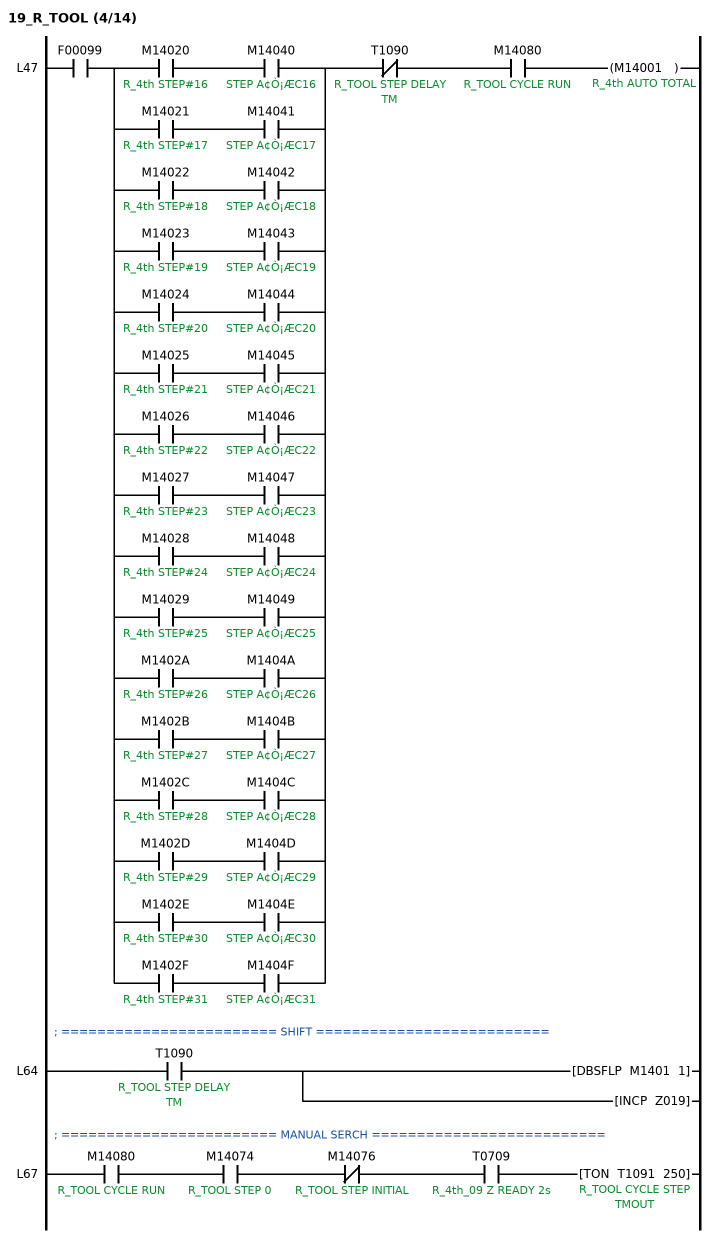
; L47
LOAD      F00099
LOAD      M14020	// R_4th STEP#16
AND       M14040	// STEP A¢Ò¡ÆC16
LOAD      M14021	// R_4th STEP#17
AND       M14041	// STEP A¢Ò¡ÆC17
OR LOAD
LOAD      M14022	// R_4th STEP#18
AND       M14042	// STEP A¢Ò¡ÆC18
OR LOAD
LOAD      M14023	// R_4th STEP#19
AND       M14043	// STEP A¢Ò¡ÆC19
OR LOAD
LOAD      M14024	// R_4th STEP#20
AND       M14044	// STEP A¢Ò¡ÆC20
OR LOAD
LOAD      M14025	// R_4th STEP#21
AND       M14045	// STEP A¢Ò¡ÆC21
OR LOAD
LOAD      M14026	// R_4th STEP#22
AND       M14046	// STEP A¢Ò¡ÆC22
OR LOAD
LOAD      M14027	// R_4th STEP#23
AND       M14047	// STEP A¢Ò¡ÆC23
OR LOAD
LOAD      M14028	// R_4th STEP#24
AND       M14048	// STEP A¢Ò¡ÆC24
OR LOAD
LOAD      M14029	// R_4th STEP#25
AND       M14049	// STEP A¢Ò¡ÆC25
OR LOAD
LOAD      M1402A	// R_4th STEP#26
AND       M1404A	// STEP A¢Ò¡ÆC26
OR LOAD
LOAD      M1402B	// R_4th STEP#27
AND       M1404B	// STEP A¢Ò¡ÆC27
OR LOAD
LOAD      M1402C	// R_4th STEP#28
AND       M1404C	// STEP A¢Ò¡ÆC28
OR LOAD
LOAD      M1402D	// R_4th STEP#29
AND       M1404D	// STEP A¢Ò¡ÆC29
OR LOAD
LOAD      M1402E	// R_4th STEP#30
AND       M1404E	// STEP A¢Ò¡ÆC30
OR LOAD
LOAD      M1402F	// R_4th STEP#31
AND       M1404F	// STEP A¢Ò¡ÆC31
OR LOAD
AND LOAD
AND NOT   T1090	// R_TOOL STEP DELAY TM
AND       M14080	// R_TOOL CYCLE RUN
OUT       M14001	// R_4th AUTO TOTAL
// ======================== SHIFT ==========================
; L64
LOAD      T1090	// R_TOOL STEP DELAY TM
DBSFLP    M1401 1
INCP      Z019
// ======================== MANUAL SERCH ==========================
; L67
LOAD      M14080	// R_TOOL CYCLE RUN
AND       M14074	// R_TOOL STEP 0
AND NOT   M14076	// R_TOOL STEP INITIAL
AND       T0709	// R_4th_09 Z READY 2s
TON       T1091 250	// R_TOOL CYCLE STEP TMOUT

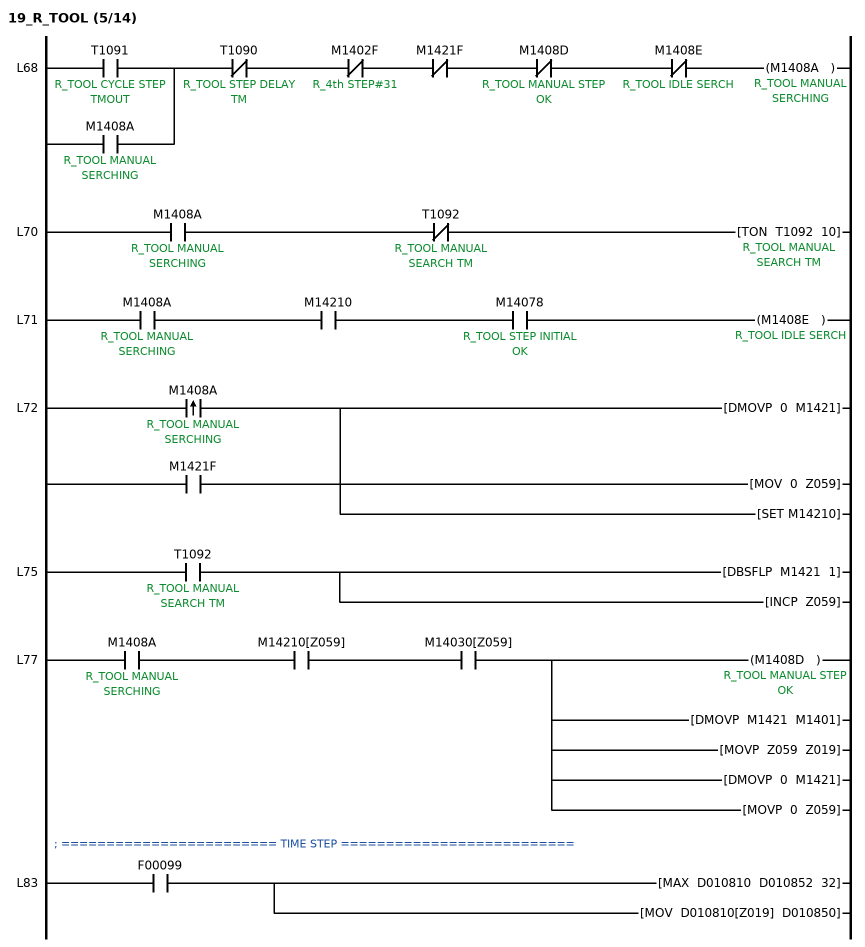
; L68
LOAD      T1091	// R_TOOL CYCLE STEP TMOUT
OR        M1408A	// R_TOOL MANUAL SERCHING
AND NOT   T1090	// R_TOOL STEP DELAY TM
AND NOT   M1402F	// R_4th STEP#31
AND NOT   M1421F
AND NOT   M1408D	// R_TOOL MANUAL STEP OK
AND NOT   M1408E	// R_TOOL IDLE SERCH
OUT       M1408A	// R_TOOL MANUAL SERCHING
; L70
LOAD      M1408A	// R_TOOL MANUAL SERCHING
AND NOT   T1092	// R_TOOL MANUAL SEARCH TM
TON       T1092 10	// R_TOOL MANUAL SEARCH TM
; L71
LOAD      M1408A	// R_TOOL MANUAL SERCHING
AND       M14210
AND       M14078	// R_TOOL STEP INITIAL OK
OUT       M1408E	// R_TOOL IDLE SERCH
; L72
LOADP     M1408A	// R_TOOL MANUAL SERCHING
OR        M1421F
DMOVP     0 M1421
MOV       0 Z059
SET       M14210
; L75
LOAD      T1092	// R_TOOL MANUAL SEARCH TM
DBSFLP    M1421 1
INCP      Z059
; L77
LOAD      M1408A	// R_TOOL MANUAL SERCHING
AND       M14210[Z059]
AND       M14030[Z059]
OUT       M1408D	// R_TOOL MANUAL STEP OK
DMOVP     M1421 M1401
MOVP      Z059 Z019
DMOVP     0 M1421
MOVP      0 Z059
// ======================== TIME STEP ==========================
; L83
LOAD      F00099
MAX       D010810 D010852 32
MOV       D010810[Z019] D010850

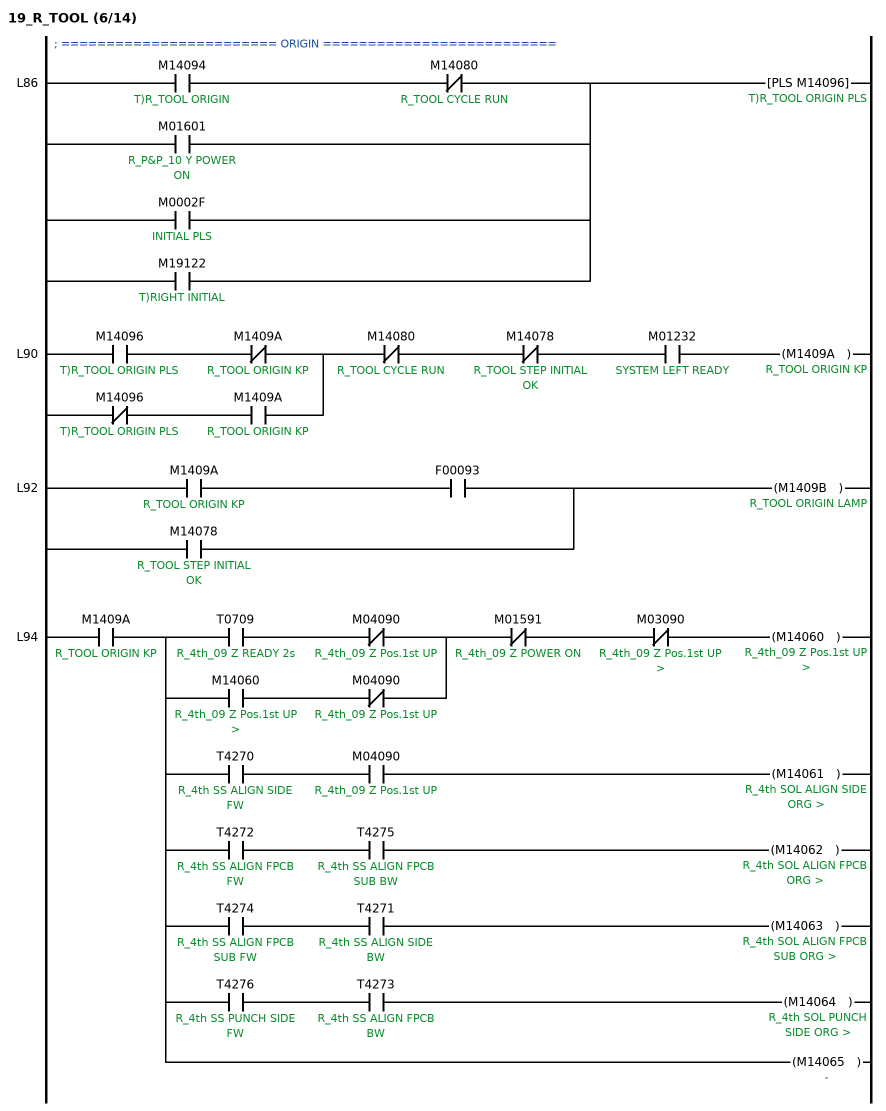
// ======================== ORIGIN ==========================
; L86
LOAD      M14094	// T)R_TOOL ORIGIN
AND NOT   M14080	// R_TOOL CYCLE RUN
OR        M01601	// R_P&P_10 Y POWER ON
OR        M0002F	// INITIAL PLS
OR        M19122	// T)RIGHT INITIAL
OUTP      M14096	// T)R_TOOL ORIGIN PLS
; L90
LOAD      M14096	// T)R_TOOL ORIGIN PLS
AND NOT   M1409A	// R_TOOL ORIGIN KP
LOAD NOT  M14096	// T)R_TOOL ORIGIN PLS
AND       M1409A	// R_TOOL ORIGIN KP
OR LOAD
AND NOT   M14080	// R_TOOL CYCLE RUN
AND NOT   M14078	// R_TOOL STEP INITIAL OK
AND       M01232	// SYSTEM LEFT READY
OUT       M1409A	// R_TOOL ORIGIN KP
; L92
LOAD      M1409A	// R_TOOL ORIGIN KP
AND       F00093
OR        M14078	// R_TOOL STEP INITIAL OK
OUT       M1409B	// R_TOOL ORIGIN LAMP
; L94
LOAD      M1409A	// R_TOOL ORIGIN KP
MPUSH
LOAD      T0709	// R_4th_09 Z READY 2s
AND NOT   M04090	// R_4th_09 Z Pos.1st UP
LOAD      M14060	// R_4th_09 Z Pos.1st UP >
AND NOT   M04090	// R_4th_09 Z Pos.1st UP
OR LOAD
AND LOAD
AND NOT   M01591	// R_4th_09 Z POWER ON
AND NOT   M03090	// R_4th_09 Z Pos.1st UP >
OUT       M14060	// R_4th_09 Z Pos.1st UP >
MLOAD
AND       T4270	// R_4th SS ALIGN SIDE FW
AND       M04090	// R_4th_09 Z Pos.1st UP
OUT       M14061	// R_4th SOL ALIGN SIDE ORG >
MLOAD
AND       T4272	// R_4th SS ALIGN FPCB FW
AND       T4275	// R_4th SS ALIGN FPCB SUB BW
OUT       M14062	// R_4th SOL ALIGN FPCB ORG >
MLOAD
AND       T4274	// R_4th SS ALIGN FPCB SUB FW
AND       T4271	// R_4th SS ALIGN SIDE BW
OUT       M14063	// R_4th SOL ALIGN FPCB SUB ORG >
MLOAD
AND       T4276	// R_4th SS PUNCH SIDE FW
AND       T4273	// R_4th SS ALIGN FPCB BW
OUT       M14064	// R_4th SOL PUNCH SIDE ORG >
MPOP
OUT       M14065	// -

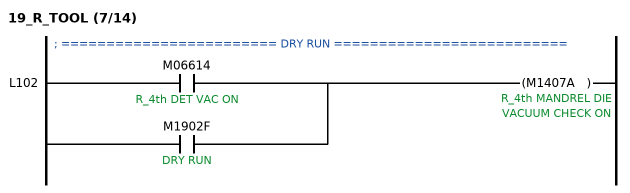
// ======================== DRY RUN ==========================
; L102
LOAD      M06614	// R_4th DET VAC ON
OR        M1902F	// DRY RUN
OUT       M1407A	// R_4th MANDREL DIE VACUUM CHECK ON

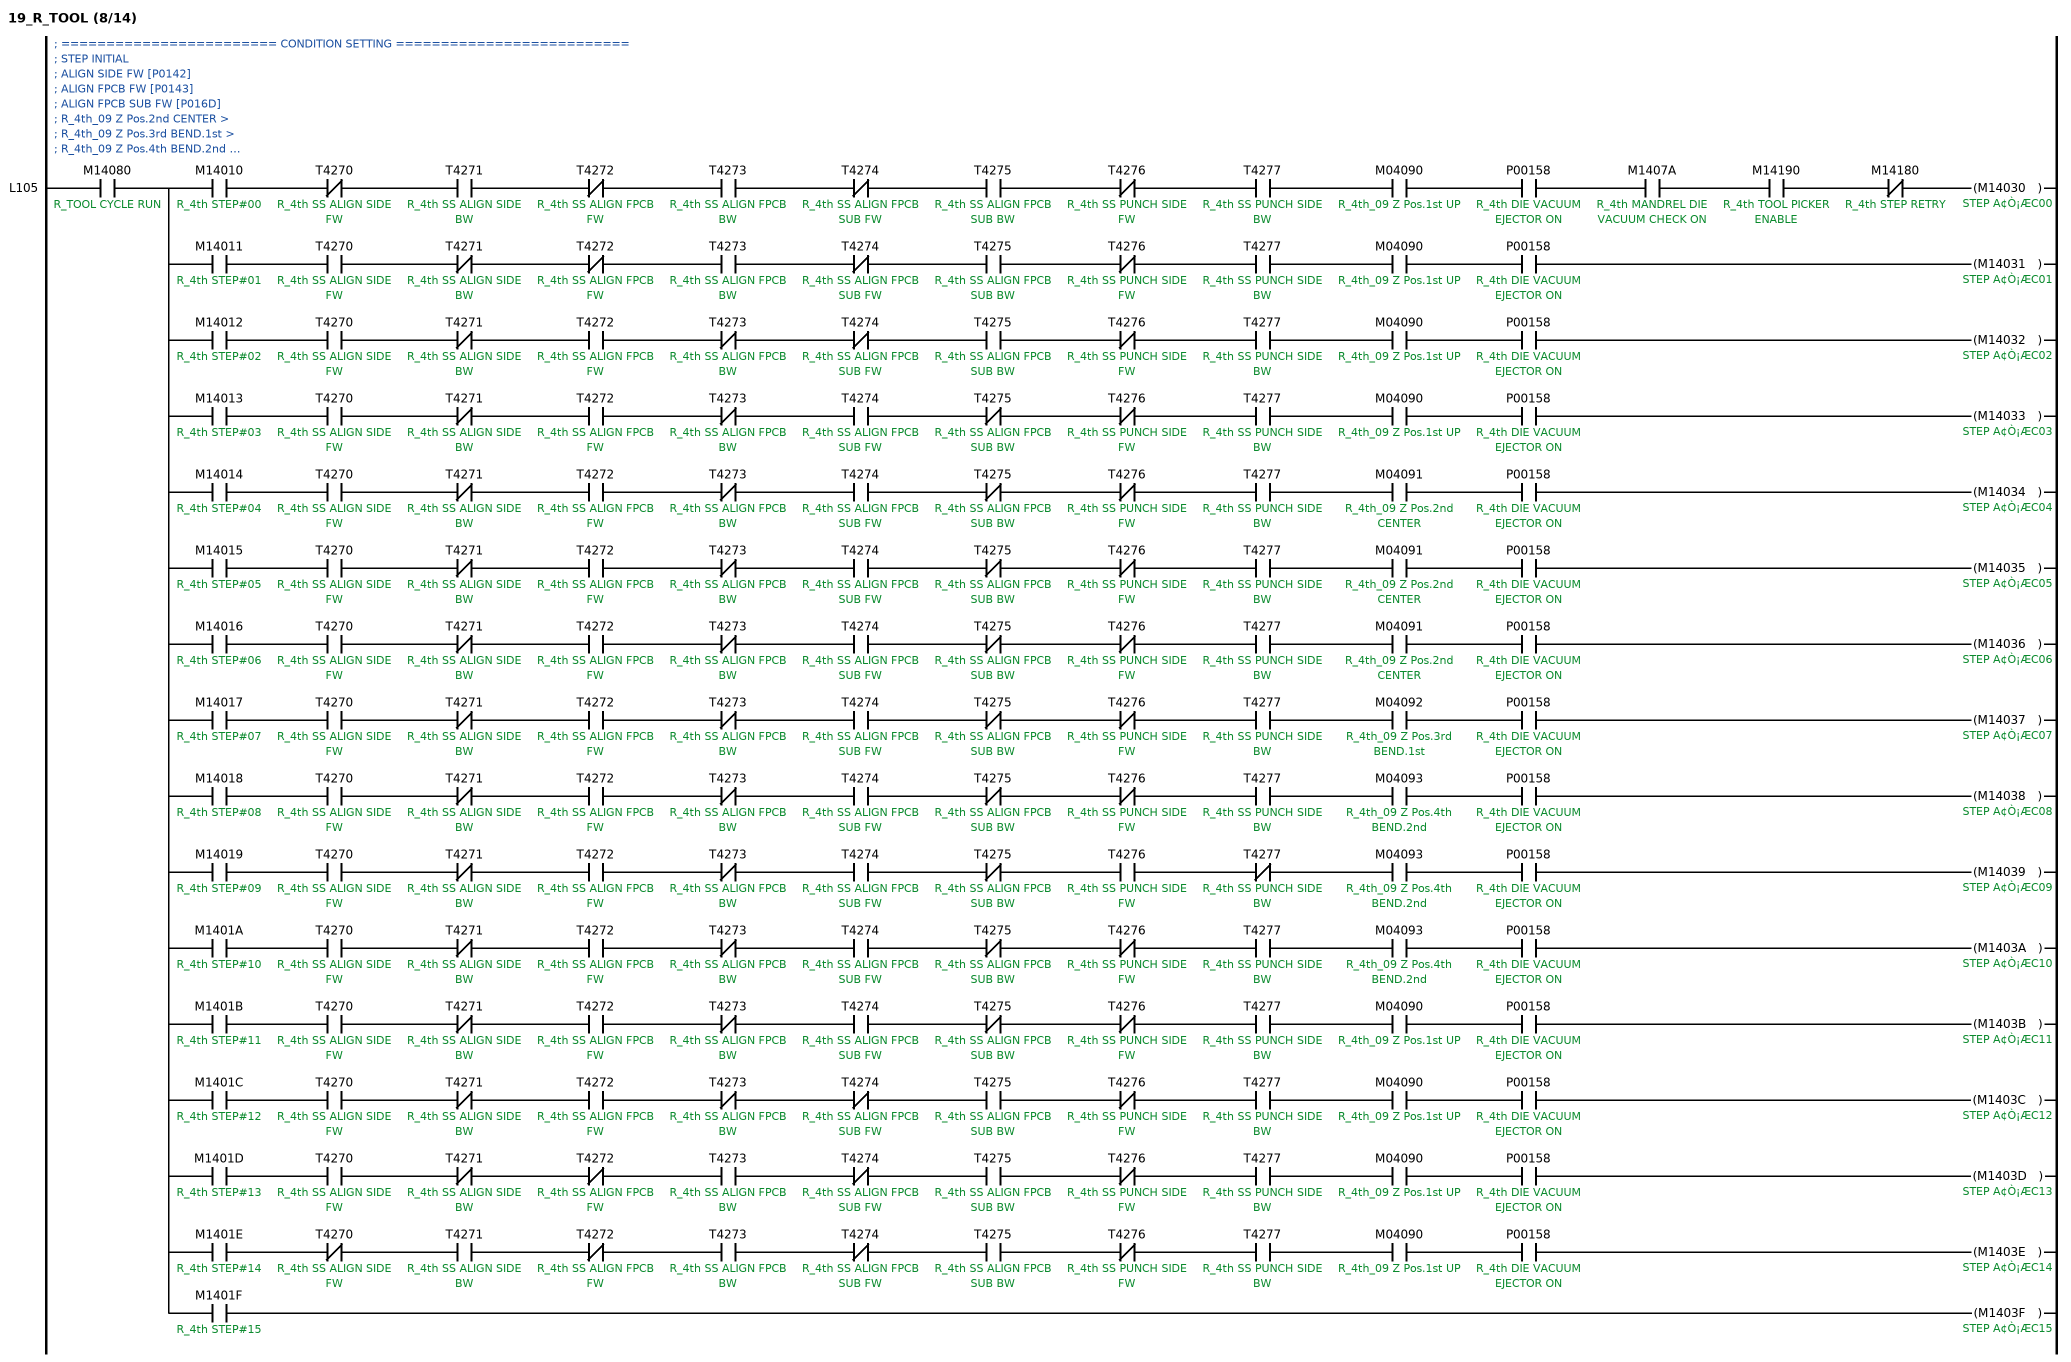
// ======================== CONDITION SETTING ==========================
; L105
LOAD      M14080	// R_TOOL CYCLE RUN
MPUSH
AND       M14010	// R_4th STEP#00
AND NOT   T4270	// R_4th SS ALIGN SIDE FW
AND       T4271	// R_4th SS ALIGN SIDE BW
AND NOT   T4272	// R_4th SS ALIGN FPCB FW
AND       T4273	// R_4th SS ALIGN FPCB BW
AND NOT   T4274	// R_4th SS ALIGN FPCB SUB FW
AND       T4275	// R_4th SS ALIGN FPCB SUB BW
AND NOT   T4276	// R_4th SS PUNCH SIDE FW
AND       T4277	// R_4th SS PUNCH SIDE BW
AND       M04090	// R_4th_09 Z Pos.1st UP
AND       P00158	// R_4th DIE VACUUM EJECTOR ON
AND       M1407A	// R_4th MANDREL DIE VACUUM CHECK ON
AND       M14190	// R_4th TOOL PICKER ENABLE
AND NOT   M14180	// R_4th STEP RETRY
OUT       M14030	// STEP A¢Ò¡ÆC00
MLOAD
AND       M14011	// R_4th STEP#01
AND       T4270	// R_4th SS ALIGN SIDE FW
AND NOT   T4271	// R_4th SS ALIGN SIDE BW
AND NOT   T4272	// R_4th SS ALIGN FPCB FW
AND       T4273	// R_4th SS ALIGN FPCB BW
AND NOT   T4274	// R_4th SS ALIGN FPCB SUB FW
AND       T4275	// R_4th SS ALIGN FPCB SUB BW
AND NOT   T4276	// R_4th SS PUNCH SIDE FW
AND       T4277	// R_4th SS PUNCH SIDE BW
AND       M04090	// R_4th_09 Z Pos.1st UP
AND       P00158	// R_4th DIE VACUUM EJECTOR ON
OUT       M14031	// STEP A¢Ò¡ÆC01
MLOAD
AND       M14012	// R_4th STEP#02
AND       T4270	// R_4th SS ALIGN SIDE FW
AND NOT   T4271	// R_4th SS ALIGN SIDE BW
AND       T4272	// R_4th SS ALIGN FPCB FW
AND NOT   T4273	// R_4th SS ALIGN FPCB BW
AND NOT   T4274	// R_4th SS ALIGN FPCB SUB FW
AND       T4275	// R_4th SS ALIGN FPCB SUB BW
AND NOT   T4276	// R_4th SS PUNCH SIDE FW
AND       T4277	// R_4th SS PUNCH SIDE BW
AND       M04090	// R_4th_09 Z Pos.1st UP
AND       P00158	// R_4th DIE VACUUM EJECTOR ON
OUT       M14032	// STEP A¢Ò¡ÆC02
MLOAD
AND       M14013	// R_4th STEP#03
AND       T4270	// R_4th SS ALIGN SIDE FW
AND NOT   T4271	// R_4th SS ALIGN SIDE BW
AND       T4272	// R_4th SS ALIGN FPCB FW
AND NOT   T4273	// R_4th SS ALIGN FPCB BW
AND       T4274	// R_4th SS ALIGN FPCB SUB FW
AND NOT   T4275	// R_4th SS ALIGN FPCB SUB BW
AND NOT   T4276	// R_4th SS PUNCH SIDE FW
AND       T4277	// R_4th SS PUNCH SIDE BW
AND       M04090	// R_4th_09 Z Pos.1st UP
AND       P00158	// R_4th DIE VACUUM EJECTOR ON
OUT       M14033	// STEP A¢Ò¡ÆC03
MLOAD
AND       M14014	// R_4th STEP#04
AND       T4270	// R_4th SS ALIGN SIDE FW
AND NOT   T4271	// R_4th SS ALIGN SIDE BW
AND       T4272	// R_4th SS ALIGN FPCB FW
AND NOT   T4273	// R_4th SS ALIGN FPCB BW
AND       T4274	// R_4th SS ALIGN FPCB SUB FW
AND NOT   T4275	// R_4th SS ALIGN FPCB SUB BW
AND NOT   T4276	// R_4th SS PUNCH SIDE FW
AND       T4277	// R_4th SS PUNCH SIDE BW
AND       M04091	// R_4th_09 Z Pos.2nd CENTER
AND       P00158	// R_4th DIE VACUUM EJECTOR ON
OUT       M14034	// STEP A¢Ò¡ÆC04
MLOAD
AND       M14015	// R_4th STEP#05
AND       T4270	// R_4th SS ALIGN SIDE FW
AND NOT   T4271	// R_4th SS ALIGN SIDE BW
AND       T4272	// R_4th SS ALIGN FPCB FW
AND NOT   T4273	// R_4th SS ALIGN FPCB BW
AND       T4274	// R_4th SS ALIGN FPCB SUB FW
AND NOT   T4275	// R_4th SS ALIGN FPCB SUB BW
AND NOT   T4276	// R_4th SS PUNCH SIDE FW
AND       T4277	// R_4th SS PUNCH SIDE BW
AND       M04091	// R_4th_09 Z Pos.2nd CENTER
AND       P00158	// R_4th DIE VACUUM EJECTOR ON
OUT       M14035	// STEP A¢Ò¡ÆC05
MLOAD
AND       M14016	// R_4th STEP#06
AND       T4270	// R_4th SS ALIGN SIDE FW
AND NOT   T4271	// R_4th SS ALIGN SIDE BW
AND       T4272	// R_4th SS ALIGN FPCB FW
AND NOT   T4273	// R_4th SS ALIGN FPCB BW
AND       T4274	// R_4th SS ALIGN FPCB SUB FW
AND NOT   T4275	// R_4th SS ALIGN FPCB SUB BW
AND NOT   T4276	// R_4th SS PUNCH SIDE FW
AND       T4277	// R_4th SS PUNCH SIDE BW
AND       M04091	// R_4th_09 Z Pos.2nd CENTER
AND       P00158	// R_4th DIE VACUUM EJECTOR ON
OUT       M14036	// STEP A¢Ò¡ÆC06
MLOAD
AND       M14017	// R_4th STEP#07
AND       T4270	// R_4th SS ALIGN SIDE FW
AND NOT   T4271	// R_4th SS ALIGN SIDE BW
AND       T4272	// R_4th SS ALIGN FPCB FW
AND NOT   T4273	// R_4th SS ALIGN FPCB BW
AND       T4274	// R_4th SS ALIGN FPCB SUB FW
AND NOT   T4275	// R_4th SS ALIGN FPCB SUB BW
AND NOT   T4276	// R_4th SS PUNCH SIDE FW
AND       T4277	// R_4th SS PUNCH SIDE BW
AND       M04092	// R_4th_09 Z Pos.3rd BEND.1st
AND       P00158	// R_4th DIE VACUUM EJECTOR ON
OUT       M14037	// STEP A¢Ò¡ÆC07
MLOAD
AND       M14018	// R_4th STEP#08
AND       T4270	// R_4th SS ALIGN SIDE FW
AND NOT   T4271	// R_4th SS ALIGN SIDE BW
AND       T4272	// R_4th SS ALIGN FPCB FW
AND NOT   T4273	// R_4th SS ALIGN FPCB BW
AND       T4274	// R_4th SS ALIGN FPCB SUB FW
AND NOT   T4275	// R_4th SS ALIGN FPCB SUB BW
AND NOT   T4276	// R_4th SS PUNCH SIDE FW
AND       T4277	// R_4th SS PUNCH SIDE BW
AND       M04093	// R_4th_09 Z Pos.4th BEND.2nd
AND       P00158	// R_4th DIE VACUUM EJECTOR ON
OUT       M14038	// STEP A¢Ò¡ÆC08
MLOAD
AND       M14019	// R_4th STEP#09
AND       T4270	// R_4th SS ALIGN SIDE FW
AND NOT   T4271	// R_4th SS ALIGN SIDE BW
AND       T4272	// R_4th SS ALIGN FPCB FW
AND NOT   T4273	// R_4th SS ALIGN FPCB BW
AND       T4274	// R_4th SS ALIGN FPCB SUB FW
AND NOT   T4275	// R_4th SS ALIGN FPCB SUB BW
AND       T4276	// R_4th SS PUNCH SIDE FW
AND NOT   T4277	// R_4th SS PUNCH SIDE BW
AND       M04093	// R_4th_09 Z Pos.4th BEND.2nd
AND       P00158	// R_4th DIE VACUUM EJECTOR ON
OUT       M14039	// STEP A¢Ò¡ÆC09
MLOAD
AND       M1401A	// R_4th STEP#10
AND       T4270	// R_4th SS ALIGN SIDE FW
AND NOT   T4271	// R_4th SS ALIGN SIDE BW
AND       T4272	// R_4th SS ALIGN FPCB FW
AND NOT   T4273	// R_4th SS ALIGN FPCB BW
AND       T4274	// R_4th SS ALIGN FPCB SUB FW
AND NOT   T4275	// R_4th SS ALIGN FPCB SUB BW
AND NOT   T4276	// R_4th SS PUNCH SIDE FW
AND       T4277	// R_4th SS PUNCH SIDE BW
AND       M04093	// R_4th_09 Z Pos.4th BEND.2nd
AND       P00158	// R_4th DIE VACUUM EJECTOR ON
OUT       M1403A	// STEP A¢Ò¡ÆC10
MLOAD
AND       M1401B	// R_4th STEP#11
AND       T4270	// R_4th SS ALIGN SIDE FW
AND NOT   T4271	// R_4th SS ALIGN SIDE BW
AND       T4272	// R_4th SS ALIGN FPCB FW
AND NOT   T4273	// R_4th SS ALIGN FPCB BW
AND       T4274	// R_4th SS ALIGN FPCB SUB FW
AND NOT   T4275	// R_4th SS ALIGN FPCB SUB BW
AND NOT   T4276	// R_4th SS PUNCH SIDE FW
AND       T4277	// R_4th SS PUNCH SIDE BW
AND       M04090	// R_4th_09 Z Pos.1st UP
AND       P00158	// R_4th DIE VACUUM EJECTOR ON
OUT       M1403B	// STEP A¢Ò¡ÆC11
MLOAD
AND       M1401C	// R_4th STEP#12
AND       T4270	// R_4th SS ALIGN SIDE FW
AND NOT   T4271	// R_4th SS ALIGN SIDE BW
AND       T4272	// R_4th SS ALIGN FPCB FW
AND NOT   T4273	// R_4th SS ALIGN FPCB BW
AND NOT   T4274	// R_4th SS ALIGN FPCB SUB FW
AND       T4275	// R_4th SS ALIGN FPCB SUB BW
AND NOT   T4276	// R_4th SS PUNCH SIDE FW
AND       T4277	// R_4th SS PUNCH SIDE BW
AND       M04090	// R_4th_09 Z Pos.1st UP
AND       P00158	// R_4th DIE VACUUM EJECTOR ON
OUT       M1403C	// STEP A¢Ò¡ÆC12
MLOAD
AND       M1401D	// R_4th STEP#13
AND       T4270	// R_4th SS ALIGN SIDE FW
AND NOT   T4271	// R_4th SS ALIGN SIDE BW
AND NOT   T4272	// R_4th SS ALIGN FPCB FW
AND       T4273	// R_4th SS ALIGN FPCB BW
AND NOT   T4274	// R_4th SS ALIGN FPCB SUB FW
AND       T4275	// R_4th SS ALIGN FPCB SUB BW
AND NOT   T4276	// R_4th SS PUNCH SIDE FW
AND       T4277	// R_4th SS PUNCH SIDE BW
AND       M04090	// R_4th_09 Z Pos.1st UP
AND       P00158	// R_4th DIE VACUUM EJECTOR ON
OUT       M1403D	// STEP A¢Ò¡ÆC13
MLOAD
AND       M1401E	// R_4th STEP#14
AND NOT   T4270	// R_4th SS ALIGN SIDE FW
AND       T4271	// R_4th SS ALIGN SIDE BW
AND NOT   T4272	// R_4th SS ALIGN FPCB FW
AND       T4273	// R_4th SS ALIGN FPCB BW
AND NOT   T4274	// R_4th SS ALIGN FPCB SUB FW
AND       T4275	// R_4th SS ALIGN FPCB SUB BW
AND NOT   T4276	// R_4th SS PUNCH SIDE FW
AND       T4277	// R_4th SS PUNCH SIDE BW
AND       M04090	// R_4th_09 Z Pos.1st UP
AND       P00158	// R_4th DIE VACUUM EJECTOR ON
OUT       M1403E	// STEP A¢Ò¡ÆC14
MPOP
AND       M1401F	// R_4th STEP#15
OUT       M1403F	// STEP A¢Ò¡ÆC15
// output comment: STEP INITIAL
// output comment: ALIGN SIDE FW [P0142]
// output comment: ALIGN FPCB FW [P0143]
// output comment: ALIGN FPCB SUB FW [P016D]
// output comment: R_4th_09 Z Pos.2nd CENTER >
// output comment: R_4th_09 Z Pos.3rd BEND.1st >
// output comment: R_4th_09 Z Pos.4th BEND.2nd >
// output comment: PUNCH SIDE FW [P016E]
// output comment: PUNCH SIDE BW [P016E]
// output comment: R_4th_09 Z Pos.1st       UP >
// output comment: ALIGN FPCB SUB BW [P016D]
// output comment: ALIGN FPCB BW [P0143]
// output comment: ALIGN SIDE BW   [P0142]

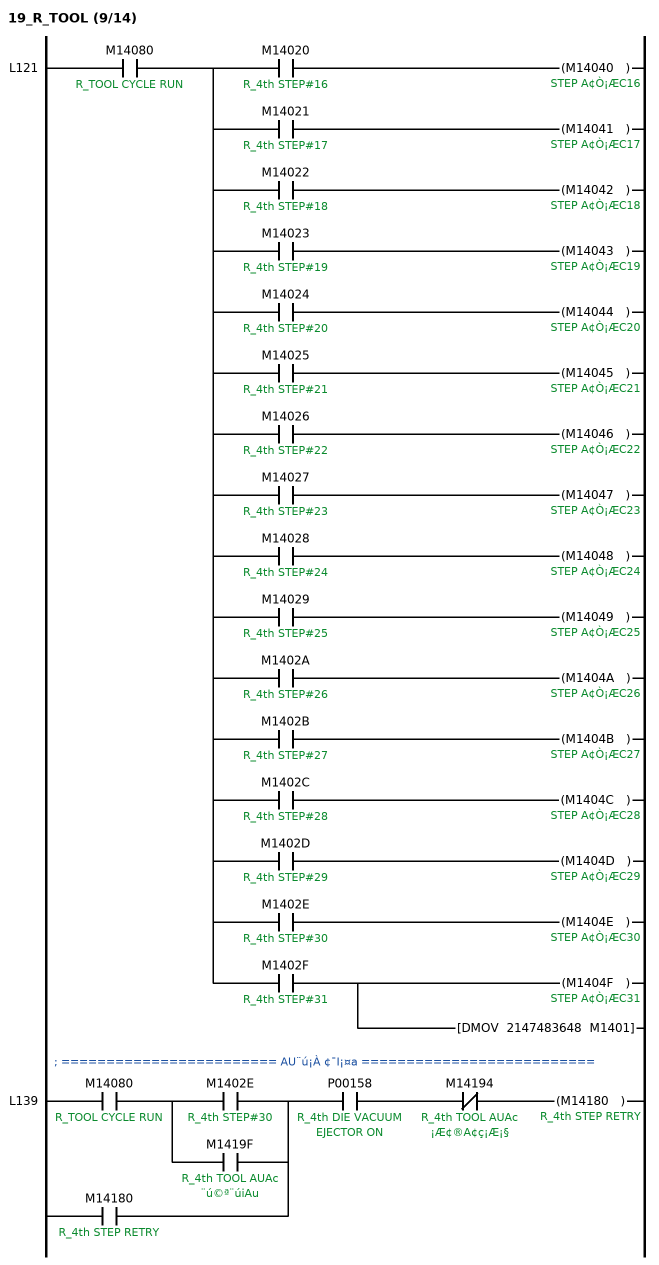
; L121
LOAD      M14080	// R_TOOL CYCLE RUN
MPUSH
AND       M14020	// R_4th STEP#16
OUT       M14040	// STEP A¢Ò¡ÆC16
MLOAD
AND       M14021	// R_4th STEP#17
OUT       M14041	// STEP A¢Ò¡ÆC17
MLOAD
AND       M14022	// R_4th STEP#18
OUT       M14042	// STEP A¢Ò¡ÆC18
MLOAD
AND       M14023	// R_4th STEP#19
OUT       M14043	// STEP A¢Ò¡ÆC19
MLOAD
AND       M14024	// R_4th STEP#20
OUT       M14044	// STEP A¢Ò¡ÆC20
MLOAD
AND       M14025	// R_4th STEP#21
OUT       M14045	// STEP A¢Ò¡ÆC21
MLOAD
AND       M14026	// R_4th STEP#22
OUT       M14046	// STEP A¢Ò¡ÆC22
MLOAD
AND       M14027	// R_4th STEP#23
OUT       M14047	// STEP A¢Ò¡ÆC23
MLOAD
AND       M14028	// R_4th STEP#24
OUT       M14048	// STEP A¢Ò¡ÆC24
MLOAD
AND       M14029	// R_4th STEP#25
OUT       M14049	// STEP A¢Ò¡ÆC25
MLOAD
AND       M1402A	// R_4th STEP#26
OUT       M1404A	// STEP A¢Ò¡ÆC26
MLOAD
AND       M1402B	// R_4th STEP#27
OUT       M1404B	// STEP A¢Ò¡ÆC27
MLOAD
AND       M1402C	// R_4th STEP#28
OUT       M1404C	// STEP A¢Ò¡ÆC28
MLOAD
AND       M1402D	// R_4th STEP#29
OUT       M1404D	// STEP A¢Ò¡ÆC29
MLOAD
AND       M1402E	// R_4th STEP#30
OUT       M1404E	// STEP A¢Ò¡ÆC30
MPOP
AND       M1402F	// R_4th STEP#31
OUT       M1404F	// STEP A¢Ò¡ÆC31
DMOV      2147483648 M1401
// ======================== AU¨ú¡À ¢¯I¡¤a ==========================
; L139
LOAD      M14080	// R_TOOL CYCLE RUN
LOAD      M1402E	// R_4th STEP#30
OR        M1419F	// R_4th TOOL AUAc ¨ú©ª¨úiAu
AND LOAD
OR        M14180	// R_4th STEP RETRY
AND       P00158	// R_4th DIE VACUUM EJECTOR ON
AND NOT   M14194	// R_4th TOOL AUAc ¡Æ¢®A¢ç¡Æ¡§
OUT       M14180	// R_4th STEP RETRY

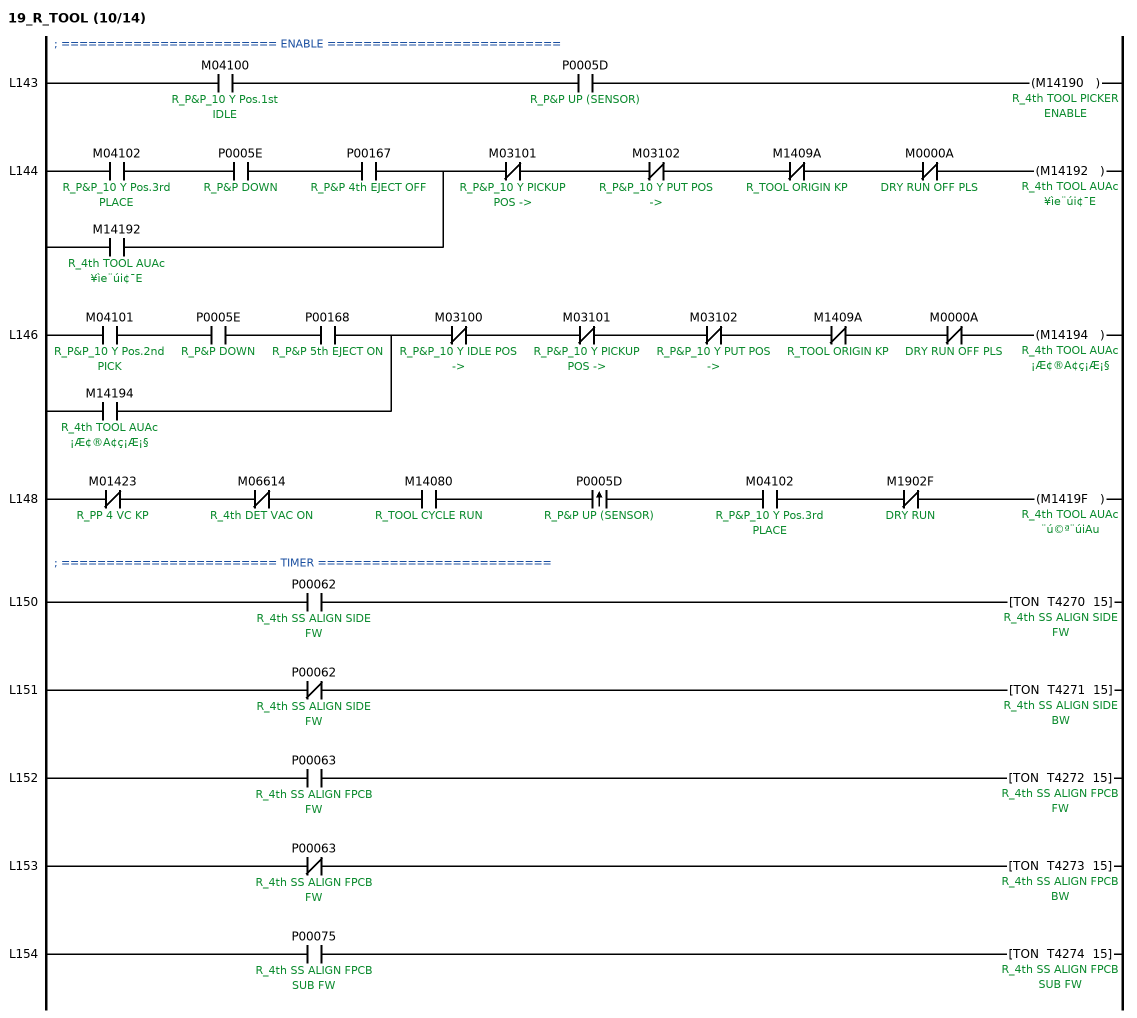
// ======================== ENABLE ==========================
; L143
LOAD      M04100	// R_P&P_10 Y Pos.1st IDLE
AND       P0005D	// R_P&P UP (SENSOR)
OUT       M14190	// R_4th TOOL PICKER ENABLE
; L144
LOAD      M04102	// R_P&P_10 Y Pos.3rd PLACE
AND       P0005E	// R_P&P DOWN
AND       P00167	// R_P&P 4th EJECT OFF
OR        M14192	// R_4th TOOL AUAc ¥ìe¨úi¢¯E
AND NOT   M03101	// R_P&P_10 Y PICKUP POS ->
AND NOT   M03102	// R_P&P_10 Y PUT POS ->
AND NOT   M1409A	// R_TOOL ORIGIN KP
AND NOT   M0000A	// DRY RUN OFF PLS
OUT       M14192	// R_4th TOOL AUAc ¥ìe¨úi¢¯E
; L146
LOAD      M04101	// R_P&P_10 Y Pos.2nd PICK
AND       P0005E	// R_P&P DOWN
AND       P00168	// R_P&P 5th EJECT ON
OR        M14194	// R_4th TOOL AUAc ¡Æ¢®A¢ç¡Æ¡§
AND NOT   M03100	// R_P&P_10 Y IDLE POS ->
AND NOT   M03101	// R_P&P_10 Y PICKUP POS ->
AND NOT   M03102	// R_P&P_10 Y PUT POS ->
AND NOT   M1409A	// R_TOOL ORIGIN KP
AND NOT   M0000A	// DRY RUN OFF PLS
OUT       M14194	// R_4th TOOL AUAc ¡Æ¢®A¢ç¡Æ¡§
; L148
LOAD NOT  M01423	// R_PP 4 VC KP
AND NOT   M06614	// R_4th DET VAC ON
AND       M14080	// R_TOOL CYCLE RUN
ANDP      P0005D	// R_P&P UP (SENSOR)
AND       M04102	// R_P&P_10 Y Pos.3rd PLACE
AND NOT   M1902F	// DRY RUN
OUT       M1419F	// R_4th TOOL AUAc ¨ú©ª¨úiAu
// ======================== TIMER ==========================
; L150
LOAD      P00062	// R_4th SS ALIGN SIDE FW
TON       T4270 15	// R_4th SS ALIGN SIDE FW
; L151
LOAD NOT  P00062	// R_4th SS ALIGN SIDE FW
TON       T4271 15	// R_4th SS ALIGN SIDE BW
; L152
LOAD      P00063	// R_4th SS ALIGN FPCB FW
TON       T4272 15	// R_4th SS ALIGN FPCB FW
; L153
LOAD NOT  P00063	// R_4th SS ALIGN FPCB FW
TON       T4273 15	// R_4th SS ALIGN FPCB BW
; L154
LOAD      P00075	// R_4th SS ALIGN FPCB SUB FW
TON       T4274 15	// R_4th SS ALIGN FPCB SUB FW

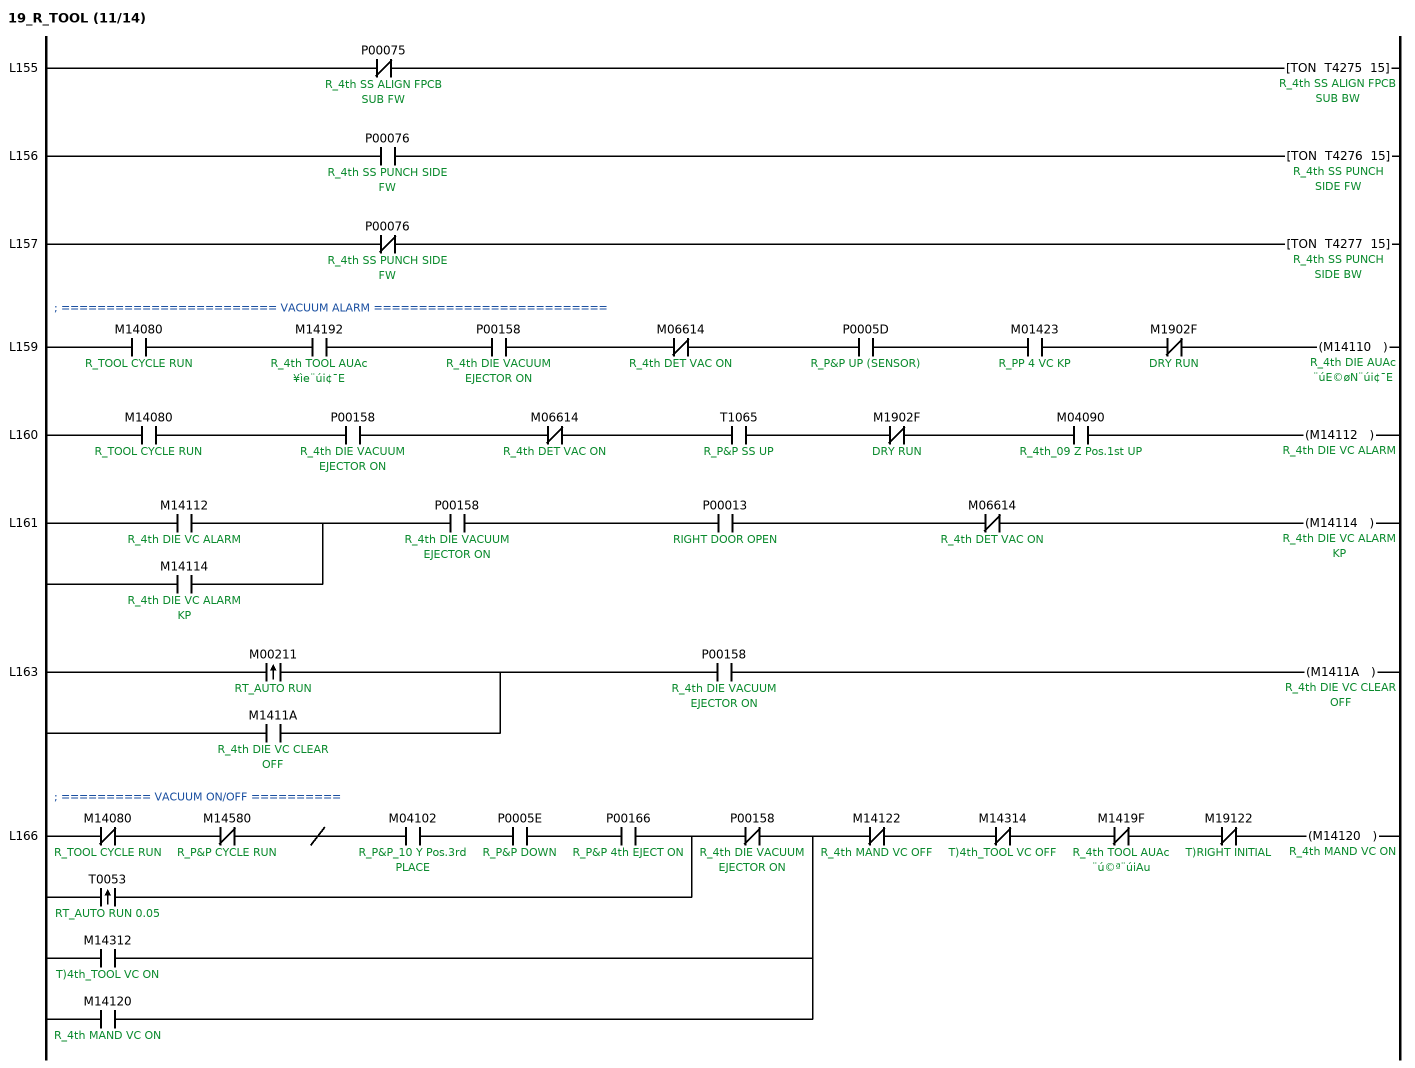
; L155
LOAD NOT  P00075	// R_4th SS ALIGN FPCB SUB FW
TON       T4275 15	// R_4th SS ALIGN FPCB SUB BW
; L156
LOAD      P00076	// R_4th SS PUNCH SIDE FW
TON       T4276 15	// R_4th SS PUNCH SIDE FW
; L157
LOAD NOT  P00076	// R_4th SS PUNCH SIDE FW
TON       T4277 15	// R_4th SS PUNCH SIDE BW
// ======================== VACUUM ALARM ==========================
; L159
LOAD      M14080	// R_TOOL CYCLE RUN
AND       M14192	// R_4th TOOL AUAc ¥ìe¨úi¢¯E
AND       P00158	// R_4th DIE VACUUM EJECTOR ON
AND NOT   M06614	// R_4th DET VAC ON
AND       P0005D	// R_P&P UP (SENSOR)
AND       M01423	// R_PP 4 VC KP
AND NOT   M1902F	// DRY RUN
OUT       M14110	// R_4th DIE AUAc ¨úE©øN¨úi¢¯E
; L160
LOAD      M14080	// R_TOOL CYCLE RUN
AND       P00158	// R_4th DIE VACUUM EJECTOR ON
AND NOT   M06614	// R_4th DET VAC ON
AND       T1065	// R_P&P SS UP
AND NOT   M1902F	// DRY RUN
AND       M04090	// R_4th_09 Z Pos.1st UP
OUT       M14112	// R_4th DIE VC ALARM
; L161
LOAD      M14112	// R_4th DIE VC ALARM
OR        M14114	// R_4th DIE VC ALARM KP
AND       P00158	// R_4th DIE VACUUM EJECTOR ON
AND       P00013	// RIGHT DOOR OPEN
AND NOT   M06614	// R_4th DET VAC ON
OUT       M14114	// R_4th DIE VC ALARM KP
; L163
LOADP     M00211	// RT_AUTO RUN
OR        M1411A	// R_4th DIE VC CLEAR OFF
AND       P00158	// R_4th DIE VACUUM EJECTOR ON
OUT       M1411A	// R_4th DIE VC CLEAR OFF
// ========== VACUUM ON/OFF ==========
; L166
LOAD NOT  M14080	// R_TOOL CYCLE RUN
AND NOT   M14580	// R_P&P CYCLE RUN
NOT
AND       M04102	// R_P&P_10 Y Pos.3rd PLACE
AND       P0005E	// R_P&P DOWN
AND       P00166	// R_P&P 4th EJECT ON
ORP       T0053	// RT_AUTO RUN 0.05
AND NOT   P00158	// R_4th DIE VACUUM EJECTOR ON
OR        M14312	// T)4th_TOOL VC ON
OR        M14120	// R_4th MAND VC ON
AND NOT   M14122	// R_4th MAND VC OFF
AND NOT   M14314	// T)4th_TOOL VC OFF
AND NOT   M1419F	// R_4th TOOL AUAc ¨ú©ª¨úiAu
AND NOT   M19122	// T)RIGHT INITIAL
OUT       M14120	// R_4th MAND VC ON

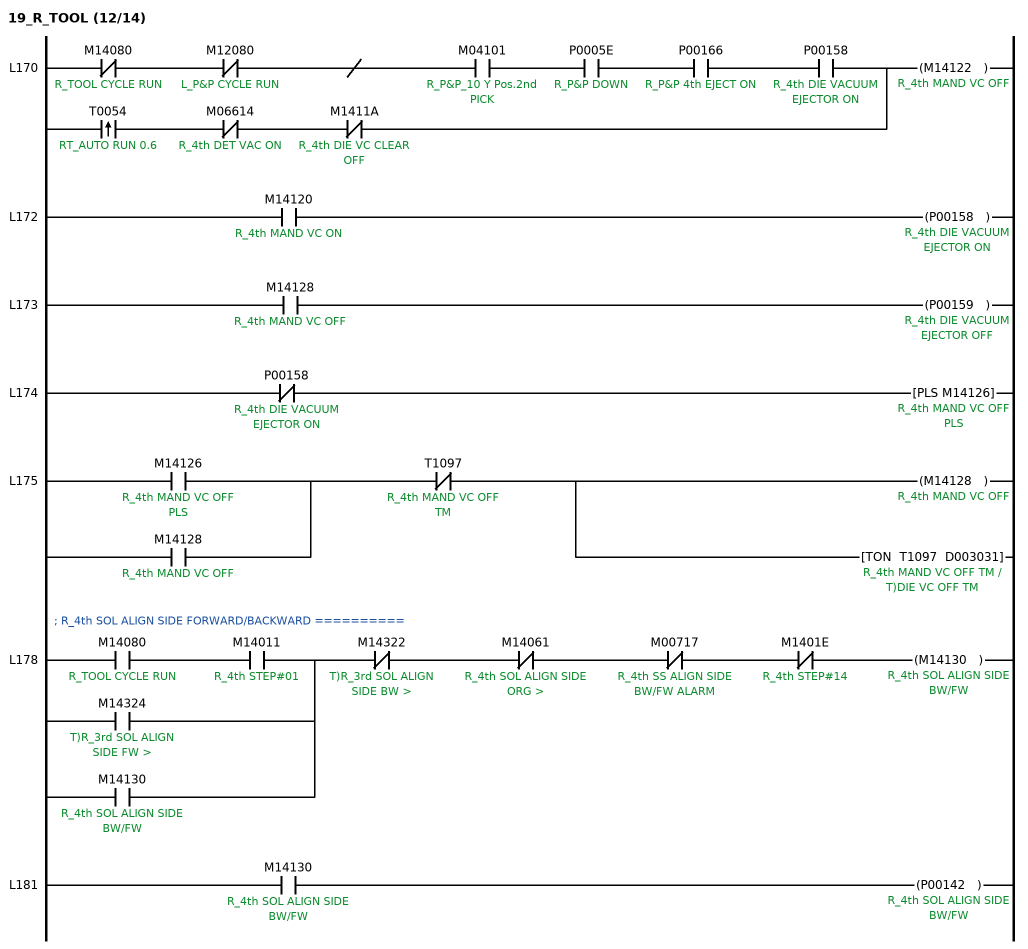
; L170
LOAD NOT  M14080	// R_TOOL CYCLE RUN
AND NOT   M12080	// L_P&P CYCLE RUN
NOT
AND       M04101	// R_P&P_10 Y Pos.2nd PICK
AND       P0005E	// R_P&P DOWN
AND       P00166	// R_P&P 4th EJECT ON
AND       P00158	// R_4th DIE VACUUM EJECTOR ON
LOADP     T0054	// RT_AUTO RUN 0.6
AND NOT   M06614	// R_4th DET VAC ON
AND NOT   M1411A	// R_4th DIE VC CLEAR OFF
OR LOAD
OUT       M14122	// R_4th MAND VC OFF
; L172
LOAD      M14120	// R_4th MAND VC ON
OUT       P00158	// R_4th DIE VACUUM EJECTOR ON
; L173
LOAD      M14128	// R_4th MAND VC OFF
OUT       P00159	// R_4th DIE VACUUM EJECTOR OFF
; L174
LOAD NOT  P00158	// R_4th DIE VACUUM EJECTOR ON
OUTP      M14126	// R_4th MAND VC OFF PLS
; L175
LOAD      M14126	// R_4th MAND VC OFF PLS
OR        M14128	// R_4th MAND VC OFF
AND NOT   T1097	// R_4th MAND VC OFF TM
OUT       M14128	// R_4th MAND VC OFF
TON       T1097 D003031	// R_4th MAND VC OFF TM / T)DIE VC OFF TM
// R_4th SOL ALIGN SIDE FORWARD/BACKWARD ==========
; L178
LOAD      M14080	// R_TOOL CYCLE RUN
AND       M14011	// R_4th STEP#01
OR        M14324	// T)R_3rd SOL ALIGN SIDE FW >
OR        M14130	// R_4th SOL ALIGN SIDE BW/FW
AND NOT   M14322	// T)R_3rd SOL ALIGN SIDE BW >
AND NOT   M14061	// R_4th SOL ALIGN SIDE ORG >
AND NOT   M00717	// R_4th SS ALIGN SIDE BW/FW ALARM
AND NOT   M1401E	// R_4th STEP#14
OUT       M14130	// R_4th SOL ALIGN SIDE BW/FW
; L181
LOAD      M14130	// R_4th SOL ALIGN SIDE BW/FW
OUT       P00142	// R_4th SOL ALIGN SIDE BW/FW

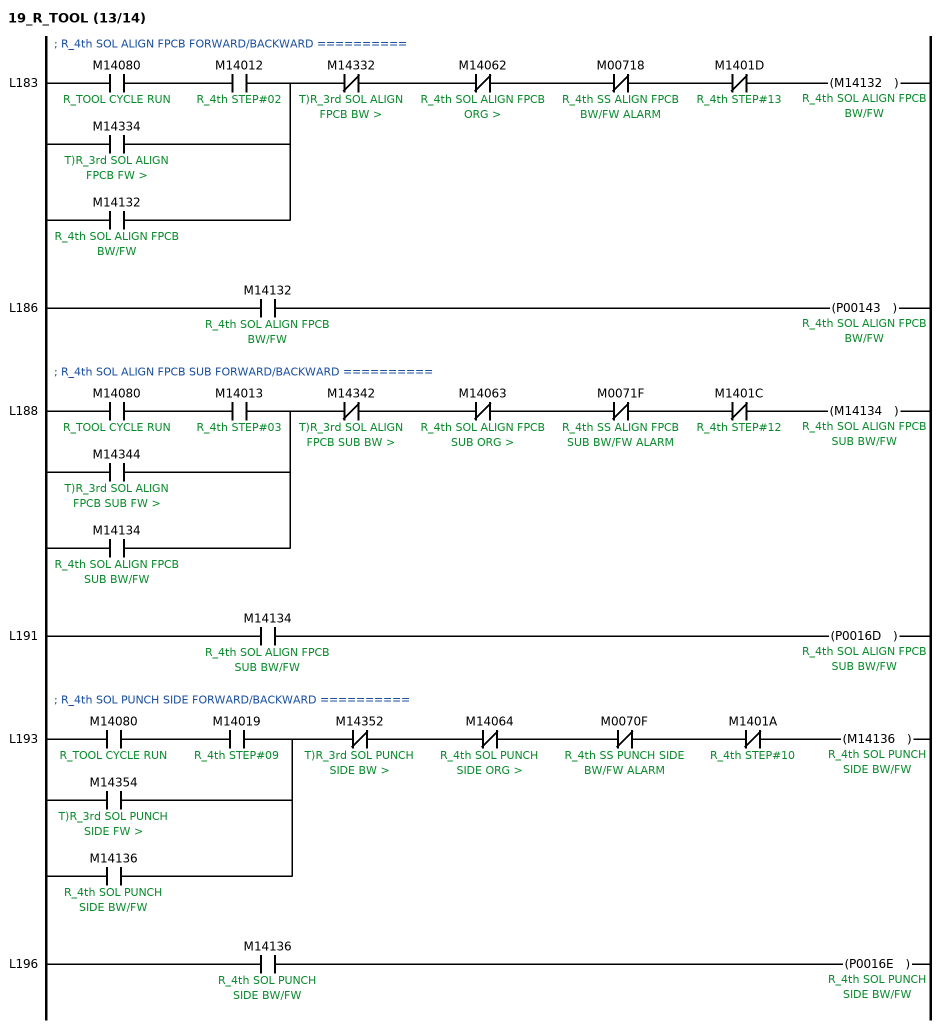
// R_4th SOL ALIGN FPCB FORWARD/BACKWARD ==========
; L183
LOAD      M14080	// R_TOOL CYCLE RUN
AND       M14012	// R_4th STEP#02
OR        M14334	// T)R_3rd SOL ALIGN FPCB FW >
OR        M14132	// R_4th SOL ALIGN FPCB BW/FW
AND NOT   M14332	// T)R_3rd SOL ALIGN FPCB BW >
AND NOT   M14062	// R_4th SOL ALIGN FPCB ORG >
AND NOT   M00718	// R_4th SS ALIGN FPCB BW/FW ALARM
AND NOT   M1401D	// R_4th STEP#13
OUT       M14132	// R_4th SOL ALIGN FPCB BW/FW
; L186
LOAD      M14132	// R_4th SOL ALIGN FPCB BW/FW
OUT       P00143	// R_4th SOL ALIGN FPCB BW/FW
// R_4th SOL ALIGN FPCB SUB FORWARD/BACKWARD ==========
; L188
LOAD      M14080	// R_TOOL CYCLE RUN
AND       M14013	// R_4th STEP#03
OR        M14344	// T)R_3rd SOL ALIGN FPCB SUB FW >
OR        M14134	// R_4th SOL ALIGN FPCB SUB BW/FW
AND NOT   M14342	// T)R_3rd SOL ALIGN FPCB SUB BW >
AND NOT   M14063	// R_4th SOL ALIGN FPCB SUB ORG >
AND NOT   M0071F	// R_4th SS ALIGN FPCB SUB BW/FW ALARM
AND NOT   M1401C	// R_4th STEP#12
OUT       M14134	// R_4th SOL ALIGN FPCB SUB BW/FW
; L191
LOAD      M14134	// R_4th SOL ALIGN FPCB SUB BW/FW
OUT       P0016D	// R_4th SOL ALIGN FPCB SUB BW/FW
// R_4th SOL PUNCH SIDE FORWARD/BACKWARD ==========
; L193
LOAD      M14080	// R_TOOL CYCLE RUN
AND       M14019	// R_4th STEP#09
OR        M14354	// T)R_3rd SOL PUNCH SIDE FW >
OR        M14136	// R_4th SOL PUNCH SIDE BW/FW
AND NOT   M14352	// T)R_3rd SOL PUNCH SIDE BW >
AND NOT   M14064	// R_4th SOL PUNCH SIDE ORG >
AND NOT   M0070F	// R_4th SS PUNCH SIDE BW/FW ALARM
AND NOT   M1401A	// R_4th STEP#10
OUT       M14136	// R_4th SOL PUNCH SIDE BW/FW
; L196
LOAD      M14136	// R_4th SOL PUNCH SIDE BW/FW
OUT       P0016E	// R_4th SOL PUNCH SIDE BW/FW

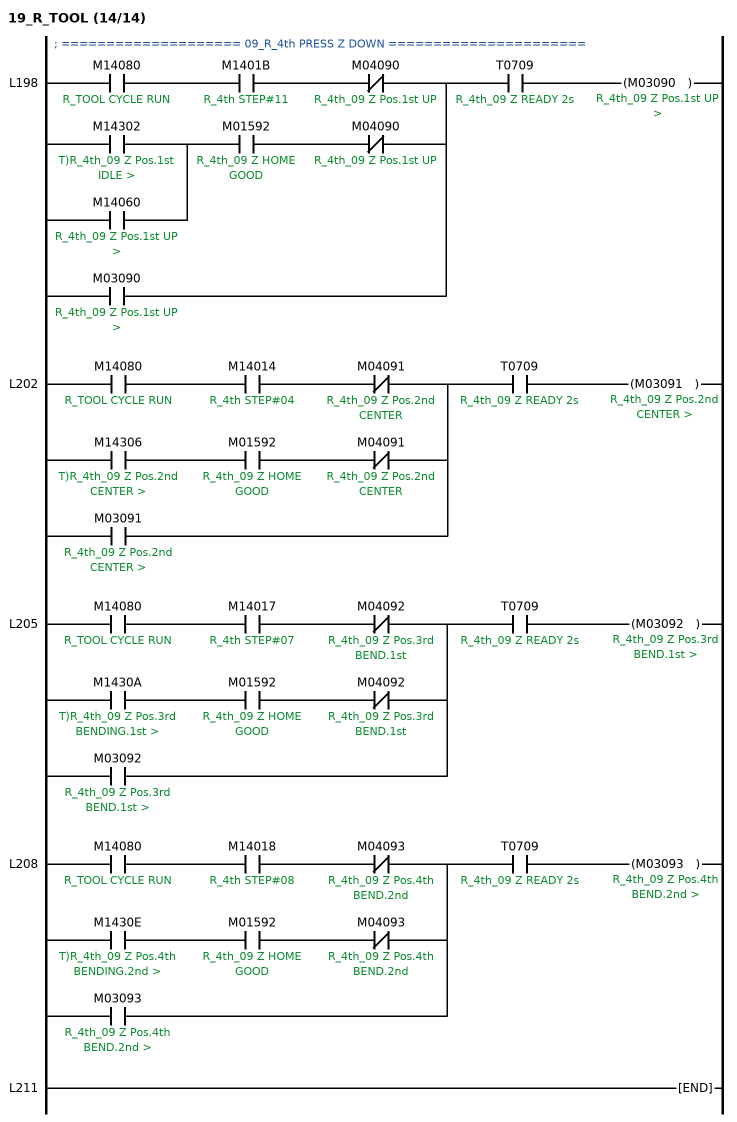
// ==================== 09_R_4th PRESS Z DOWN ======================
; L198
LOAD      M14080	// R_TOOL CYCLE RUN
AND       M1401B	// R_4th STEP#11
AND NOT   M04090	// R_4th_09 Z Pos.1st UP
LOAD      M14302	// T)R_4th_09 Z Pos.1st IDLE >
OR        M14060	// R_4th_09 Z Pos.1st UP >
AND       M01592	// R_4th_09 Z HOME GOOD
AND NOT   M04090	// R_4th_09 Z Pos.1st UP
OR LOAD
OR        M03090	// R_4th_09 Z Pos.1st UP >
AND       T0709	// R_4th_09 Z READY 2s
OUT       M03090	// R_4th_09 Z Pos.1st UP >
; L202
LOAD      M14080	// R_TOOL CYCLE RUN
AND       M14014	// R_4th STEP#04
AND NOT   M04091	// R_4th_09 Z Pos.2nd CENTER
LOAD      M14306	// T)R_4th_09 Z Pos.2nd CENTER >
AND       M01592	// R_4th_09 Z HOME GOOD
AND NOT   M04091	// R_4th_09 Z Pos.2nd CENTER
OR LOAD
OR        M03091	// R_4th_09 Z Pos.2nd CENTER >
AND       T0709	// R_4th_09 Z READY 2s
OUT       M03091	// R_4th_09 Z Pos.2nd CENTER >
; L205
LOAD      M14080	// R_TOOL CYCLE RUN
AND       M14017	// R_4th STEP#07
AND NOT   M04092	// R_4th_09 Z Pos.3rd BEND.1st
LOAD      M1430A	// T)R_4th_09 Z Pos.3rd BENDING.1st >
AND       M01592	// R_4th_09 Z HOME GOOD
AND NOT   M04092	// R_4th_09 Z Pos.3rd BEND.1st
OR LOAD
OR        M03092	// R_4th_09 Z Pos.3rd BEND.1st >
AND       T0709	// R_4th_09 Z READY 2s
OUT       M03092	// R_4th_09 Z Pos.3rd BEND.1st >
; L208
LOAD      M14080	// R_TOOL CYCLE RUN
AND       M14018	// R_4th STEP#08
AND NOT   M04093	// R_4th_09 Z Pos.4th BEND.2nd
LOAD      M1430E	// T)R_4th_09 Z Pos.4th BENDING.2nd >
AND       M01592	// R_4th_09 Z HOME GOOD
AND NOT   M04093	// R_4th_09 Z Pos.4th BEND.2nd
OR LOAD
OR        M03093	// R_4th_09 Z Pos.4th BEND.2nd >
AND       T0709	// R_4th_09 Z READY 2s
OUT       M03093	// R_4th_09 Z Pos.4th BEND.2nd >
; L211
END

PROGRAM 20_R_PP (task: ¨ö¨¬A¥ì CA¡¤I¡¾¡¿¡¤¡Í)

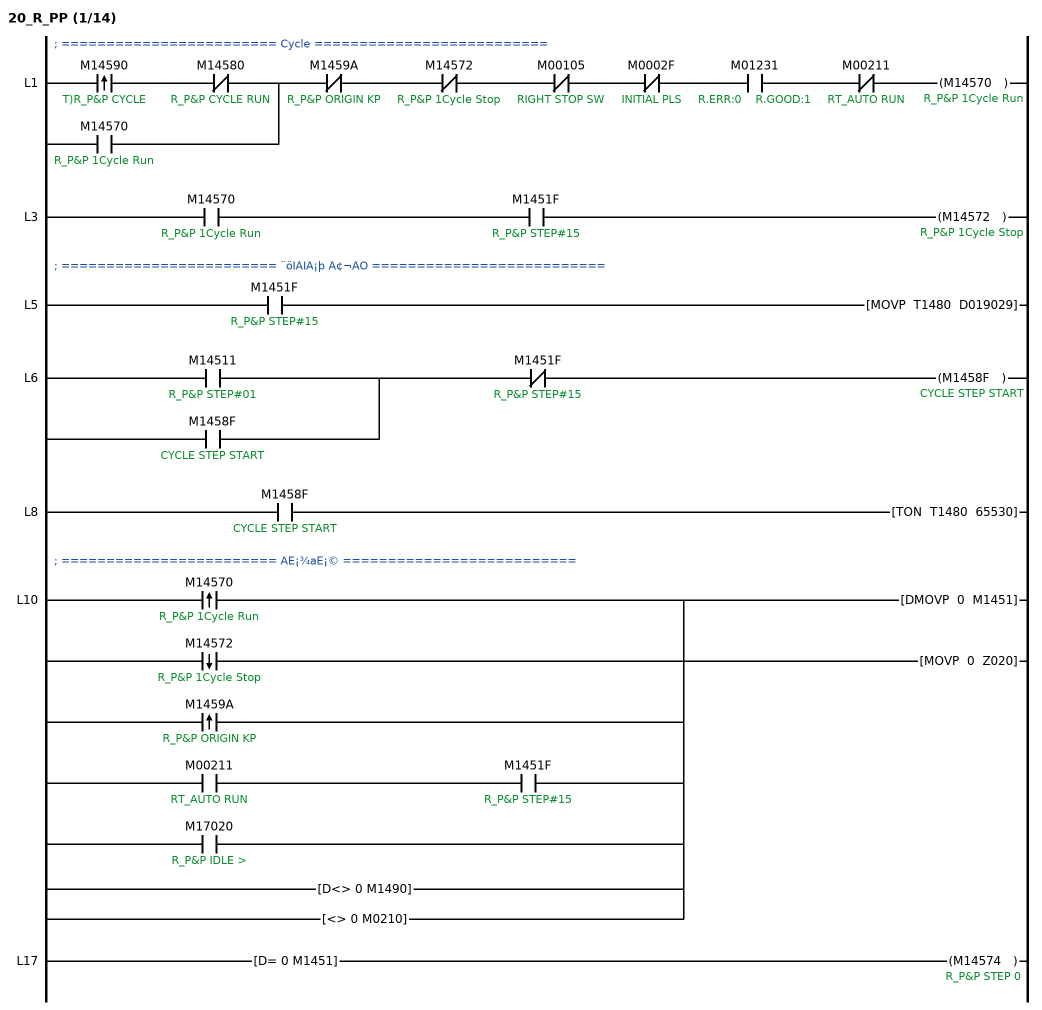
// ======================== Cycle ==========================
; L1
LOADP     M14590	// T)R_P&P CYCLE
AND NOT   M14580	// R_P&P CYCLE RUN
OR        M14570	// R_P&P 1Cycle Run
AND NOT   M1459A	// R_P&P ORIGIN KP
AND NOT   M14572	// R_P&P 1Cycle Stop
AND NOT   M00105	// RIGHT STOP SW
AND NOT   M0002F	// INITIAL PLS
AND       M01231	// R.ERR:0    R.GOOD:1
AND NOT   M00211	// RT_AUTO RUN
OUT       M14570	// R_P&P 1Cycle Run
; L3
LOAD      M14570	// R_P&P 1Cycle Run
AND       M1451F	// R_P&P STEP#15
OUT       M14572	// R_P&P 1Cycle Stop
// ======================== ¨öIAIA¡þ A¢¬AO ==========================
; L5
LOAD      M1451F	// R_P&P STEP#15
MOVP      T1480 D019029
; L6
LOAD      M14511	// R_P&P STEP#01
OR        M1458F	// CYCLE STEP START
AND NOT   M1451F	// R_P&P STEP#15
OUT       M1458F	// CYCLE STEP START
; L8
LOAD      M1458F	// CYCLE STEP START
TON       T1480 65530
// ======================== AE¡¾aE¡© ==========================
; L10
LOADP     M14570	// R_P&P 1Cycle Run
ORN       M14572	// R_P&P 1Cycle Stop
ORP       M1459A	// R_P&P ORIGIN KP
LOAD      M00211	// RT_AUTO RUN
AND       M1451F	// R_P&P STEP#15
OR LOAD
OR        M17020	// R_P&P IDLE >
ORD<>     0 M1490
OR<>      0 M0210
DMOVP     0 M1451
MOVP      0 Z020
; L17
LOADD=    0 M1451
OUT       M14574	// R_P&P STEP 0

